LIN {X 0,Y 288.96,Z 785.854,A -85,B 0,C 180,E1 8748.983,E2 8748.983} C_VEL
LIN {X 0,Y 289.698,Z 782.109,A -85,B 0,C 180,E1 8744.907,E2 8744.907} C_VEL
LIN {X 0,Y 291.072,Z 776.715,A -85,B 0,C 180,E1 8740.892,E2 8740.892} C_VEL
LIN {X 0,Y 293.159,Z 769.854,A -85,B 0,C 180,E1 8737.044,E2 8737.044} C_VEL
LIN {X 0,Y 296.063,Z 761.342,A -85,B 0,C 180,E1 8733.293,E2 8733.293} C_VEL
LIN {X 0,Y 299.636,Z 751.536,A -85,B 0,C 180,E1 8729.811,E2 8729.811} C_VEL
LIN {X 0,Y 304.006,Z 739.719,A -85,B 0,C 180,E1 8726.419,E2 8726.419} C_VEL
LIN {X 0,Y 308.871,Z 726.48,A -85,B 0,C 180,E1 8723.31,E2 8723.31} C_VEL
LIN {X 0,Y 314.092,Z 711.806,A -85,B 0,C 180,E1 8720.474,E2 8720.474} C_VEL
LIN {X 0,Y 319.545,Z 695.592,A -85,B 0,C 180,E1 8717.901,E2 8717.901} C_VEL
LIN {X 0,Y 324.669,Z 679.065,A -85,B 0,C 180,E1 8715.739,E2 8715.739} C_VEL
LIN {X 0,Y 329.752,Z 660.963,A -85,B 0,C 180,E1 8713.804,E2 8713.804} C_VEL
LIN {X 0,Y 334.408,Z 641.774,A -85,B 0,C 180,E1 8712.156,E2 8712.156} C_VEL
LIN {X 0,Y 338.298,Z 622.744,A -85,B 0,C 180,E1 8710.851,E2 8710.851} C_VEL
LIN {X 0,Y 341.828,Z 601.532,A -85,B 0,C 180,E1 8709.727,E2 8709.727} C_VEL
LIN {X 0,Y 344.554,Z 579.645,A -85,B 0,C 180,E1 8708.89,E2 8708.89} C_VEL
LIN {X 0,Y 346.384,Z 556.456,A -85,B 0,C 180,E1 8708.295,E2 8708.295} C_VEL
LIN {X 0,Y 350.037,Z 495.768,A -85,B 0,C 180,E1 8706.999,E2 8706.999} C_VEL
LIN {X 0,Y 349.833,Z 488.203,A -85,B 0,C 180,E1 8706.711,E2 8706.711} C_VEL
LIN {X 0,Y 347.018,Z 468.467,A -85,B 0,C 180,E1 8705.501,E2 8705.501} C_VEL
LIN {X 0,Y 346.964,Z 461.961,A -85,B 0,C 180,E1 8705.269,E2 8705.269} C_VEL
LIN {X 0,Y 352.089,Z 380.587,A -85,B 0,C 180,E1 8703.525,E2 8703.525} C_VEL
LIN {X 0,Y 342.307,Z 363.806,A -85,B 0,C 180,E1 8700.718,E2 8700.718} C_VEL
LIN {X 0,Y 333.106,Z 349.419,A -85,B 0,C 180,E1 8697.824,E2 8697.824} C_VEL
LIN {X 0,Y 323.644,Z 335.645,A -85,B 0,C 180,E1 8694.496,E2 8694.496} C_VEL
LIN {X 0,Y 316.195,Z 325.679,A -85,B 0,C 180,E1 8691.572,E2 8691.572} C_VEL
LIN {X 0,Y 312.253,Z 320.486,A -85,B 0,C 180,E1 8689.859,E2 8689.859} C_VEL
LIN {X 0,Y 307.488,Z 314.479,A -85,B 0,C 180,E1 8687.657,E2 8687.657} C_VEL
LIN {X 0,Y 303.986,Z 310.183,A -85,B 0,C 180,E1 8685.875,E2 8685.875} C_VEL
LIN {X 0,Y 299.931,Z 305.159,A -85,B 0,C 180,E1 8683.632,E2 8683.632} C_VEL
LIN {X 0,Y 296.324,Z 300.805,A -85,B 0,C 180,E1 8681.4,E2 8681.4} C_VEL
LIN {X 0,Y 295.437,Z 299.331,A -85,B 0,C 180,E1 8680.523,E2 8680.523} C_VEL
LIN {X 0,Y 293.137,Z 295.553,A -85,B 0,C 180,E1 8677.627,E2 8677.627} C_VEL
LIN {X 0,Y 292.608,Z 294.29,A -85,B 0,C 180,E1 8676.723,E2 8676.723} C_VEL
LIN {X 0,Y 289.99,Z 290.354,A -85,B 0,C 180,E1 8672.728,E2 8672.728} C_VEL
LIN {X 0,Y 289.321,Z 288.803,A -85,B 0,C 180,E1 8671.221,E2 8671.221} C_VEL
LIN {X 0,Y 286.275,Z 283.926,A -85,B 0,C 180,E1 8662.778,E2 8662.778} C_VEL
LIN {X 0,Y 285.612,Z 283.017,A -85,B 0,C 180,E1 8658.786,E2 8658.786} C_VEL
LIN {X 0,Y 285.73,Z 283.102,A -85,B 0,C 180,E1 8652.94,E2 8652.94} C_VEL
LIN {X 0,Y 286.409,Z 284.215,A -85,B 0,C 180,E1 8649.037,E2 8649.037} C_VEL
LIN {X 0,Y 289.951,Z 289.598,A -85,B 0,C 180,E1 8640.38,E2 8640.38} C_VEL
LIN {X 0,Y 292.353,Z 293.977,A -85,B 0,C 180,E1 8636.273,E2 8636.273} C_VEL
LIN {X 0,Y 293.355,Z 295.125,A -85,B 0,C 180,E1 8635.11,E2 8635.11} C_VEL
LIN {X 0,Y 295.652,Z 299.397,A -85,B 0,C 180,E1 8632.028,E2 8632.028} C_VEL
LIN {X 0,Y 296.617,Z 300.723,A -85,B 0,C 180,E1 8631.078,E2 8631.078} C_VEL
LIN {X 0,Y 300.225,Z 305.323,A -85,B 0,C 180,E1 8628.764,E2 8628.764} C_VEL
LIN {X 0,Y 302.029,Z 307.444,A -85,B 0,C 180,E1 8627.718,E2 8627.718} C_VEL
LIN {X 0,Y 306.76,Z 313.199,A -85,B 0,C 180,E1 8625.222,E2 8625.222} C_VEL
LIN {X 0,Y 311.135,Z 318.616,A -85,B 0,C 180,E1 8623.139,E2 8623.139} C_VEL
LIN {X 0,Y 315.417,Z 324.086,A -85,B 0,C 180,E1 8621.23,E2 8621.23} C_VEL
LIN {X 0,Y 322.474,Z 333.247,A -85,B 0,C 180,E1 8618.394,E2 8618.394} C_VEL
LIN {X 0,Y 332.455,Z 347.118,A -85,B 0,C 180,E1 8614.813,E2 8614.813} C_VEL
LIN {X 0,Y 343.288,Z 363.412,A -85,B 0,C 180,E1 8611.371,E2 8611.371} C_VEL
LIN {X 0,Y 353.776,Z 380.644,A -85,B 0,C 180,E1 8608.38,E2 8608.38} C_VEL
LIN {X 0,Y 356.871,Z 386.273,A -85,B 0,C 180,E1 8607.544,E2 8607.544} C_VEL
LIN {X 0,Y 344.365,Z 598.77,A -85,B 0,C 180,E1 8603.126,E2 8603.126} C_VEL
LIN {X 0,Y 341.699,Z 620.996,A -85,B 0,C 180,E1 8602.442,E2 8602.442} C_VEL
LIN {X 0,Y 338.23,Z 641.686,A -85,B 0,C 180,E1 8601.567,E2 8601.567} C_VEL
LIN {X 0,Y 334.015,Z 662.2,A -85,B 0,C 180,E1 8600.424,E2 8600.424} C_VEL
LIN {X 0,Y 329.158,Z 681.971,A -85,B 0,C 180,E1 8599.009,E2 8599.009} C_VEL
LIN {X 0,Y 323.758,Z 701.072,A -85,B 0,C 180,E1 8597.305,E2 8597.305} C_VEL
LIN {X 0,Y 317.973,Z 719.569,A -85,B 0,C 180,E1 8595.285,E2 8595.285} C_VEL
LIN {X 0,Y 311.98,Z 737.297,A -85,B 0,C 180,E1 8592.921,E2 8592.921} C_VEL
LIN {X 0,Y 305.913,Z 753.989,A -85,B 0,C 180,E1 8590.201,E2 8590.201} C_VEL
LIN {X 0,Y 300.011,Z 769.739,A -85,B 0,C 180,E1 8587.098,E2 8587.098} C_VEL
LIN {X 0,Y 294.8,Z 783.662,A -85,B 0,C 180,E1 8583.793,E2 8583.793} C_VEL
LIN {X 0,Y 290.144,Z 796.44,A -85,B 0,C 180,E1 8580.12,E2 8580.12} C_VEL
LIN {X 0,Y 286.319,Z 807.649,A -85,B 0,C 180,E1 8576.17,E2 8576.17} C_VEL
LIN {X 0,Y 283.403,Z 817.534,A -85,B 0,C 180,E1 8571.892,E2 8571.892} C_VEL
LIN {X 0,Y 281.612,Z 825.183,A -85,B 0,C 180,E1 8567.776,E2 8567.776} C_VEL
LIN {X 0,Y 280.64,Z 831.149,A -85,B 0,C 180,E1 8563.598,E2 8563.598} C_VEL
LIN {X 0,Y 280.321,Z 835.68,A -85,B 0,C 180,E1 8559.234,E2 8559.234} C_VEL
LIN {X 0,Y 280.368,Z 838.327,A -85,B 0,C 180,E1 8555.318,E2 8555.318} C_VEL
LIN {X 0,Y 280.465,Z 839.49,A -85,B 0,C 180,E1 8551.428,E2 8551.428} C_VEL
LIN {X 0,Y 280.457,Z 839.377,A -85,B 0,C 180,E1 8547.955,E2 8547.955} C_VEL
LIN {X 0,Y 280.349,Z 837.945,A -85,B 0,C 180,E1 8544.061,E2 8544.061} C_VEL
LIN {X 0,Y 280.337,Z 835.069,A -85,B 0,C 180,E1 8540.14,E2 8540.14} C_VEL
LIN {X 0,Y 280.737,Z 830.298,A -85,B 0,C 180,E1 8535.772,E2 8535.772} C_VEL
LIN {X 0,Y 281.821,Z 824.143,A -85,B 0,C 180,E1 8531.591,E2 8531.591} C_VEL
LIN {X 0,Y 283.811,Z 816.119,A -85,B 0,C 180,E1 8527.374,E2 8527.374} C_VEL
LIN {X 0,Y 286.968,Z 805.984,A -85,B 0,C 180,E1 8523.065,E2 8523.065} C_VEL
LIN {X 0,Y 290.951,Z 794.89,A -85,B 0,C 180,E1 8519.198,E2 8519.198} C_VEL
LIN {X 0,Y 296.028,Z 781.655,A -85,B 0,C 180,E1 8515.427,E2 8515.427} C_VEL
LIN {X 0,Y 301.627,Z 767.471,A -85,B 0,C 180,E1 8512.088,E2 8512.088} C_VEL
LIN {X 0,Y 308.077,Z 751.16,A -85,B 0,C 180,E1 8508.91,E2 8508.91} C_VEL
LIN {X 0,Y 314.475,Z 734.51,A -85,B 0,C 180,E1 8506.234,E2 8506.234} C_VEL
LIN {X 0,Y 320.933,Z 716.552,A -85,B 0,C 180,E1 8503.876,E2 8503.876} C_VEL
LIN {X 0,Y 327.063,Z 698.101,A -85,B 0,C 180,E1 8501.891,E2 8501.891} C_VEL
LIN {X 0,Y 332.717,Z 679.347,A -85,B 0,C 180,E1 8500.242,E2 8500.242} C_VEL
LIN {X 0,Y 338.053,Z 658.99,A -85,B 0,C 180,E1 8498.81,E2 8498.81} C_VEL
LIN {X 0,Y 342.508,Z 638.773,A -85,B 0,C 180,E1 8497.709,E2 8497.709} C_VEL
LIN {X 0,Y 346.488,Z 616.391,A -85,B 0,C 180,E1 8496.8,E2 8496.8} C_VEL
LIN {X 0,Y 349.201,Z 594.573,A -85,B 0,C 180,E1 8496.155,E2 8496.155} C_VEL
LIN {X 0,Y 363.212,Z 387.306,A -85,B 0,C 180,E1 8491.769,E2 8491.769} C_VEL
LIN {X 0,Y 357.13,Z 375.817,A -85,B 0,C 180,E1 8489.469,E2 8489.469} C_VEL
LIN {X 0,Y 351.809,Z 366.536,A -85,B 0,C 180,E1 8487.179,E2 8487.179} C_VEL
LIN {X 0,Y 346.722,Z 358.345,A -85,B 0,C 180,E1 8484.628,E2 8484.628} C_VEL
LIN {X 0,Y 342.725,Z 352.195,A -85,B 0,C 180,E1 8482.199,E2 8482.199} C_VEL
LIN {X 0,Y 338.782,Z 346.281,A -85,B 0,C 180,E1 8479.124,E2 8479.124} C_VEL
LIN {X 0,Y 335.351,Z 341.275,A -85,B 0,C 180,E1 8474.858,E2 8474.858} C_VEL
LIN {X 0,Y 334.083,Z 340.173,A -85,B 0,C 180,E1 8470.869,E2 8470.869} C_VEL
LIN {X 0,Y 334.8,Z 340.86,A -85,B 0,C 180,E1 8467.034,E2 8467.034} C_VEL
LIN {X 0,Y 335.429,Z 341.751,A -85,B 0,C 180,E1 8465.732,E2 8465.732} C_VEL
LIN {X 0,Y 338.722,Z 346.674,A -85,B 0,C 180,E1 8461.693,E2 8461.693} C_VEL
LIN {X 0,Y 342.538,Z 352.567,A -85,B 0,C 180,E1 8458.663,E2 8458.663} C_VEL
LIN {X 0,Y 346.974,Z 359.516,A -85,B 0,C 180,E1 8455.953,E2 8455.953} C_VEL
LIN {X 0,Y 351.61,Z 367.232,A -85,B 0,C 180,E1 8453.593,E2 8453.593} C_VEL
LIN {X 0,Y 357.61,Z 377.851,A -85,B 0,C 180,E1 8450.993,E2 8450.993} C_VEL
LIN {X 0,Y 361.836,Z 386.289,A -85,B 0,C 180,E1 8449.342,E2 8449.342} C_VEL
LIN {X 0,Y 347.156,Z 576.519,A -85,B 0,C 180,E1 8445.157,E2 8445.157} C_VEL
LIN {X 0,Y 344.505,Z 597.249,A -85,B 0,C 180,E1 8444.439,E2 8444.439} C_VEL
LIN {X 0,Y 341.005,Z 617.374,A -85,B 0,C 180,E1 8443.478,E2 8443.478} C_VEL
LIN {X 0,Y 336.446,Z 638.132,A -85,B 0,C 180,E1 8442.178,E2 8442.178} C_VEL
LIN {X 0,Y 331.586,Z 656.641,A -85,B 0,C 180,E1 8440.706,E2 8440.706} C_VEL
LIN {X 0,Y 325.902,Z 675.297,A -85,B 0,C 180,E1 8438.857,E2 8438.857} C_VEL
LIN {X 0,Y 319.749,Z 693.072,A -85,B 0,C 180,E1 8436.667,E2 8436.667} C_VEL
LIN {X 0,Y 313.63,Z 709.09,A -85,B 0,C 180,E1 8434.242,E2 8434.242} C_VEL
LIN {X 0,Y 307.613,Z 723.755,A -85,B 0,C 180,E1 8431.533,E2 8431.533} C_VEL
LIN {X 0,Y 301.449,Z 738.039,A -85,B 0,C 180,E1 8428.298,E2 8428.298} C_VEL
LIN {X 0,Y 296.18,Z 749.926,A -85,B 0,C 180,E1 8424.98,E2 8424.98} C_VEL
LIN {X 0,Y 291.545,Z 760.386,A -85,B 0,C 180,E1 8421.381,E2 8421.381} C_VEL
LIN {X 0,Y 287.493,Z 769.777,A -85,B 0,C 180,E1 8417.301,E2 8417.301} C_VEL
LIN {X 0,Y 284.581,Z 776.948,A -85,B 0,C 180,E1 8413.247,E2 8413.247} C_VEL
LIN {X 0,Y 282.636,Z 782.301,A -85,B 0,C 180,E1 8409.223,E2 8409.223} C_VEL
LIN {X 0,Y 281.403,Z 786.349,A -85,B 0,C 180,E1 8404.842,E2 8404.842} C_VEL
LIN {X 0,Y 280.867,Z 788.559,A -85,B 0,C 180,E1 8400.841,E2 8400.841} C_VEL
LIN {X 0,Y 280.669,Z 789.27,A -85,B 0,C 180,E1 8396.902,E2 8396.902} C_VEL
LIN {X 0,Y 280.703,Z 788.609,A -85,B 0,C 180,E1 8392.848,E2 8392.848} C_VEL
LIN {X 0,Y 281.012,Z 786.58,A -85,B 0,C 180,E1 8388.844,E2 8388.844} C_VEL
LIN {X 0,Y 281.762,Z 782.987,A -85,B 0,C 180,E1 8384.805,E2 8384.805} C_VEL
LIN {X 0,Y 283.151,Z 777.829,A -85,B 0,C 180,E1 8380.789,E2 8380.789} C_VEL
LIN {X 0,Y 285.445,Z 770.71,A -85,B 0,C 180,E1 8376.64,E2 8376.64} C_VEL
LIN {X 0,Y 288.513,Z 762.206,A -85,B 0,C 180,E1 8372.783,E2 8372.783} C_VEL
LIN {X 0,Y 292.494,Z 751.817,A -85,B 0,C 180,E1 8369.023,E2 8369.023} C_VEL
LIN {X 0,Y 297.12,Z 739.943,A -85,B 0,C 180,E1 8365.563,E2 8365.563} C_VEL
LIN {X 0,Y 302.24,Z 726.611,A -85,B 0,C 180,E1 8362.398,E2 8362.398} C_VEL
LIN {X 0,Y 307.541,Z 712.321,A -85,B 0,C 180,E1 8359.607,E2 8359.607} C_VEL
LIN {X 0,Y 313.218,Z 696.066,A -85,B 0,C 180,E1 8356.996,E2 8356.996} C_VEL
LIN {X 0,Y 318.548,Z 679.49,A -85,B 0,C 180,E1 8354.808,E2 8354.808} C_VEL
LIN {X 0,Y 323.823,Z 661.34,A -85,B 0,C 180,E1 8352.852,E2 8352.852} C_VEL
LIN {X 0,Y 328.65,Z 642.115,A -85,B 0,C 180,E1 8351.189,E2 8351.189} C_VEL
LIN {X 0,Y 332.677,Z 623.038,A -85,B 0,C 180,E1 8349.874,E2 8349.874} C_VEL
LIN {X 0,Y 336.314,Z 601.867,A -85,B 0,C 180,E1 8348.747,E2 8348.747} C_VEL
LIN {X 0,Y 339.148,Z 579.793,A -85,B 0,C 180,E1 8347.9,E2 8347.9} C_VEL
LIN {X 0,Y 341.054,Z 556.224,A -85,B 0,C 180,E1 8347.295,E2 8347.295} C_VEL
LIN {X 0,Y 346.964,Z 461.961,A -85,B 0,C 180,E1 8345.269,E2 8345.269} C_VEL
LIN {X 0,Y 346.834,Z 454.394,A -85,B 0,C 180,E1 8344.982,E2 8344.982} C_VEL
LIN {X 0,Y 344.217,Z 434.656,A -85,B 0,C 180,E1 8343.751,E2 8343.751} C_VEL
LIN {X 0,Y 344.179,Z 428.151,A -85,B 0,C 180,E1 8343.512,E2 8343.512} C_VEL
LIN {X 0,Y 346.995,Z 384.26,A -85,B 0,C 180,E1 8342.555,E2 8342.555} C_VEL
LIN {X 0,Y 337.233,Z 367.447,A -85,B 0,C 180,E1 8339.626,E2 8339.626} C_VEL
LIN {X 0,Y 328.644,Z 354.039,A -85,B 0,C 180,E1 8336.798,E2 8336.798} C_VEL
LIN {X 0,Y 320.15,Z 341.516,A -85,B 0,C 180,E1 8333.68,E2 8333.68} C_VEL
LIN {X 0,Y 313.353,Z 332.296,A -85,B 0,C 180,E1 8330.908,E2 8330.908} C_VEL
LIN {X 0,Y 309.764,Z 327.505,A -85,B 0,C 180,E1 8329.309,E2 8329.309} C_VEL
LIN {X 0,Y 304.951,Z 321.32,A -85,B 0,C 180,E1 8327.005,E2 8327.005} C_VEL
LIN {X 0,Y 301.631,Z 317.18,A -85,B 0,C 180,E1 8325.248,E2 8325.248} C_VEL
LIN {X 0,Y 297.992,Z 312.599,A -85,B 0,C 180,E1 8323.192,E2 8323.192} C_VEL
LIN {X 0,Y 294.364,Z 308.114,A -85,B 0,C 180,E1 8320.895,E2 8320.895} C_VEL
LIN {X 0,Y 292.939,Z 306.545,A -85,B 0,C 180,E1 8319.914,E2 8319.914} C_VEL
LIN {X 0,Y 289.269,Z 302.244,A -85,B 0,C 180,E1 8317.218,E2 8317.218} C_VEL
LIN {X 0,Y 288.179,Z 300.837,A -85,B 0,C 180,E1 8316.265,E2 8316.265} C_VEL
LIN {X 0,Y 285.556,Z 296.562,A -85,B 0,C 180,E1 8312.153,E2 8312.153} C_VEL
LIN {X 0,Y 284.77,Z 295.304,A -85,B 0,C 180,E1 8310.602,E2 8310.602} C_VEL
LIN {X 0,Y 282.142,Z 290.71,A -85,B 0,C 180,E1 8302.501,E2 8302.501} C_VEL
LIN {X 0,Y 281.507,Z 289.878,A -85,B 0,C 180,E1 8298.211,E2 8298.211} C_VEL
LIN {X 0,Y 281.76,Z 290.08,A -85,B 0,C 180,E1 8292.5,E2 8292.5} C_VEL
LIN {X 0,Y 282.36,Z 291.206,A -85,B 0,C 180,E1 8288.917,E2 8288.917} C_VEL
LIN {X 0,Y 285.744,Z 296.313,A -85,B 0,C 180,E1 8280.6,E2 8280.6} C_VEL
LIN {X 0,Y 288.201,Z 300.781,A -85,B 0,C 180,E1 8276.418,E2 8276.418} C_VEL
LIN {X 0,Y 289.496,Z 302.21,A -85,B 0,C 180,E1 8275.244,E2 8275.244} C_VEL
LIN {X 0,Y 293.06,Z 306.64,A -85,B 0,C 180,E1 8272.549,E2 8272.549} C_VEL
LIN {X 0,Y 294.752,Z 308.37,A -85,B 0,C 180,E1 8271.415,E2 8271.415} C_VEL
LIN {X 0,Y 298.672,Z 313.092,A -85,B 0,C 180,E1 8268.998,E2 8268.998} C_VEL
LIN {X 0,Y 304.696,Z 320.601,A -85,B 0,C 180,E1 8265.654,E2 8265.654} C_VEL
LIN {X 0,Y 308.931,Z 325.927,A -85,B 0,C 180,E1 8263.596,E2 8263.596} C_VEL
LIN {X 0,Y 313.153,Z 331.425,A -85,B 0,C 180,E1 8261.668,E2 8261.668} C_VEL
LIN {X 0,Y 319.919,Z 340.337,A -85,B 0,C 180,E1 8258.887,E2 8258.887} C_VEL
LIN {X 0,Y 329.429,Z 353.77,A -85,B 0,C 180,E1 8255.381,E2 8255.381} C_VEL
LIN {X 0,Y 339.989,Z 369.918,A -85,B 0,C 180,E1 8251.93,E2 8251.93} C_VEL
LIN {X 0,Y 350.662,Z 387.725,A -85,B 0,C 180,E1 8248.809,E2 8248.809} C_VEL
LIN {X 0,Y 351.752,Z 389.961,A -85,B 0,C 180,E1 8248.496,E2 8248.496} C_VEL
LIN {X 0,Y 339.052,Z 598.328,A -85,B 0,C 180,E1 8244.137,E2 8244.137} C_VEL
LIN {X 0,Y 336.324,Z 620.453,A -85,B 0,C 180,E1 8243.455,E2 8243.455} C_VEL
LIN {X 0,Y 332.728,Z 641.297,A -85,B 0,C 180,E1 8242.572,E2 8242.572} C_VEL
LIN {X 0,Y 328.51,Z 661.261,A -85,B 0,C 180,E1 8241.459,E2 8241.459} C_VEL
LIN {X 0,Y 323.497,Z 681.072,A -85,B 0,C 180,E1 8240.038,E2 8240.038} C_VEL
LIN {X 0,Y 317.936,Z 700.164,A -85,B 0,C 180,E1 8238.332,E2 8238.332} C_VEL
LIN {X 0,Y 311.912,Z 718.8,A -85,B 0,C 180,E1 8236.287,E2 8236.287} C_VEL
LIN {X 0,Y 305.677,Z 736.578,A -85,B 0,C 180,E1 8233.9,E2 8233.9} C_VEL
LIN {X 0,Y 299.5,Z 752.941,A -85,B 0,C 180,E1 8231.209,E2 8231.209} C_VEL
LIN {X 0,Y 293.274,Z 768.84,A -85,B 0,C 180,E1 8228.042,E2 8228.042} C_VEL
LIN {X 0,Y 287.866,Z 782.632,A -85,B 0,C 180,E1 8224.721,E2 8224.721} C_VEL
LIN {X 0,Y 283.011,Z 795.216,A -85,B 0,C 180,E1 8221.049,E2 8221.049} C_VEL
LIN {X 0,Y 278.97,Z 806.37,A -85,B 0,C 180,E1 8217.074,E2 8217.074} C_VEL
LIN {X 0,Y 275.752,Z 816.549,A -85,B 0,C 180,E1 8212.601,E2 8212.601} C_VEL
LIN {X 0,Y 273.762,Z 824.423,A -85,B 0,C 180,E1 8208.266,E2 8208.266} C_VEL
LIN {X 0,Y 272.705,Z 830.359,A -85,B 0,C 180,E1 8204.001,E2 8204.001} C_VEL
LIN {X 0,Y 272.344,Z 834.925,A -85,B 0,C 180,E1 8199.507,E2 8199.507} C_VEL
LIN {X 0,Y 272.381,Z 837.47,A -85,B 0,C 180,E1 8195.686,E2 8195.686} C_VEL
LIN {X 0,Y 272.492,Z 838.748,A -85,B 0,C 180,E1 8191.68,E2 8191.68} C_VEL
LIN {X 0,Y 272.491,Z 838.693,A -85,B 0,C 180,E1 8188.105,E2 8188.105} C_VEL
LIN {X 0,Y 272.372,Z 837.365,A -85,B 0,C 180,E1 8184.098,E2 8184.098} C_VEL
LIN {X 0,Y 272.352,Z 834.541,A -85,B 0,C 180,E1 8180.062,E2 8180.062} C_VEL
LIN {X 0,Y 272.771,Z 829.868,A -85,B 0,C 180,E1 8175.564,E2 8175.564} C_VEL
LIN {X 0,Y 273.914,Z 823.762,A -85,B 0,C 180,E1 8171.261,E2 8171.261} C_VEL
LIN {X 0,Y 276.007,Z 815.908,A -85,B 0,C 180,E1 8166.948,E2 8166.948} C_VEL
LIN {X 0,Y 279.251,Z 806.144,A -85,B 0,C 180,E1 8162.62,E2 8162.62} C_VEL
LIN {X 0,Y 283.549,Z 794.847,A -85,B 0,C 180,E1 8158.539,E2 8158.539} C_VEL
LIN {X 0,Y 288.869,Z 781.727,A -85,B 0,C 180,E1 8154.685,E2 8154.685} C_VEL
LIN {X 0,Y 294.968,Z 767.163,A -85,B 0,C 180,E1 8151.162,E2 8151.162} C_VEL
LIN {X 0,Y 301.446,Z 751.617,A -85,B 0,C 180,E1 8148.058,E2 8148.058} C_VEL
LIN {X 0,Y 308.373,Z 734.455,A -85,B 0,C 180,E1 8145.243,E2 8145.243} C_VEL
LIN {X 0,Y 315.108,Z 716.565,A -85,B 0,C 180,E1 8142.861,E2 8142.861} C_VEL
LIN {X 0,Y 321.655,Z 697.65,A -85,B 0,C 180,E1 8140.805,E2 8140.805} C_VEL
LIN {X 0,Y 327.521,Z 679.016,A -85,B 0,C 180,E1 8139.155,E2 8139.155} C_VEL
LIN {X 0,Y 333.072,Z 658.633,A -85,B 0,C 180,E1 8137.718,E2 8137.718} C_VEL
LIN {X 0,Y 337.797,Z 637.894,A -85,B 0,C 180,E1 8136.592,E2 8136.592} C_VEL
LIN {X 0,Y 341.94,Z 615.26,A -85,B 0,C 180,E1 8135.683,E2 8135.683} C_VEL
LIN {X 0,Y 344.716,Z 593.311,A -85,B 0,C 180,E1 8135.039,E2 8135.039} C_VEL
LIN {X 0,Y 358.984,Z 391.402,A -85,B 0,C 180,E1 8130.738,E2 8130.738} C_VEL
LIN {X 0,Y 353.499,Z 380.693,A -85,B 0,C 180,E1 8128.51,E2 8128.51} C_VEL
LIN {X 0,Y 347.702,Z 370.44,A -85,B 0,C 180,E1 8125.782,E2 8125.782} C_VEL
LIN {X 0,Y 342.941,Z 362.606,A -85,B 0,C 180,E1 8123.089,E2 8123.089} C_VEL
LIN {X 0,Y 339.712,Z 357.776,A -85,B 0,C 180,E1 8120.864,E2 8120.864} C_VEL
LIN {X 0,Y 337.208,Z 353.82,A -85,B 0,C 180,E1 8118.678,E2 8118.678} C_VEL
LIN {X 0,Y 334.208,Z 349.161,A -85,B 0,C 180,E1 8114.733,E2 8114.733} C_VEL
LIN {X 0,Y 333.004,Z 348.094,A -85,B 0,C 180,E1 8110.73,E2 8110.73} C_VEL
LIN {X 0,Y 333.784,Z 348.857,A -85,B 0,C 180,E1 8106.883,E2 8106.883} C_VEL
LIN {X 0,Y 334.321,Z 349.825,A -85,B 0,C 180,E1 8105.751,E2 8105.751} C_VEL
LIN {X 0,Y 337.323,Z 354.442,A -85,B 0,C 180,E1 8101.955,E2 8101.955} C_VEL
LIN {X 0,Y 341.021,Z 360.377,A -85,B 0,C 180,E1 8098.899,E2 8098.899} C_VEL
LIN {X 0,Y 345.256,Z 367.344,A -85,B 0,C 180,E1 8096.224,E2 8096.224} C_VEL
LIN {X 0,Y 349.539,Z 374.718,A -85,B 0,C 180,E1 8093.967,E2 8093.967} C_VEL
LIN {X 0,Y 355.163,Z 385.134,A -85,B 0,C 180,E1 8091.421,E2 8091.421} C_VEL
LIN {X 0,Y 357.679,Z 390.488,A -85,B 0,C 180,E1 8090.376,E2 8090.376} C_VEL
LIN {X 0,Y 342.678,Z 577.001,A -85,B 0,C 180,E1 8086.256,E2 8086.256} C_VEL
LIN {X 0,Y 339.89,Z 597.985,A -85,B 0,C 180,E1 8085.526,E2 8085.526} C_VEL
LIN {X 0,Y 336.338,Z 617.732,A -85,B 0,C 180,E1 8084.583,E2 8084.583} C_VEL
LIN {X 0,Y 331.695,Z 638.196,A -85,B 0,C 180,E1 8083.304,E2 8083.304} C_VEL
LIN {X 0,Y 326.543,Z 657.073,A -85,B 0,C 180,E1 8081.803,E2 8081.803} C_VEL
LIN {X 0,Y 320.484,Z 676.157,A -85,B 0,C 180,E1 8079.9,E2 8079.9} C_VEL
LIN {X 0,Y 314.241,Z 693.465,A -85,B 0,C 180,E1 8077.753,E2 8077.753} C_VEL
LIN {X 0,Y 307.989,Z 709.12,A -85,B 0,C 180,E1 8075.37,E2 8075.37} C_VEL
LIN {X 0,Y 301.488,Z 724.292,A -85,B 0,C 180,E1 8072.552,E2 8072.552} C_VEL
LIN {X 0,Y 295.167,Z 738.222,A -85,B 0,C 180,E1 8069.365,E2 8069.365} C_VEL
LIN {X 0,Y 289.548,Z 750.249,A -85,B 0,C 180,E1 8065.974,E2 8065.974} C_VEL
LIN {X 0,Y 284.531,Z 760.916,A -85,B 0,C 180,E1 8062.25,E2 8062.25} C_VEL
LIN {X 0,Y 280.248,Z 770.153,A -85,B 0,C 180,E1 8058.154,E2 8058.154} C_VEL
LIN {X 0,Y 277.155,Z 777.214,A -85,B 0,C 180,E1 8054.121,E2 8054.121} C_VEL
LIN {X 0,Y 274.913,Z 782.902,A -85,B 0,C 180,E1 8049.802,E2 8049.802} C_VEL
LIN {X 0,Y 273.568,Z 786.914,A -85,B 0,C 180,E1 8045.413,E2 8045.413} C_VEL
LIN {X 0,Y 272.932,Z 789.272,A -85,B 0,C 180,E1 8041.103,E2 8041.103} C_VEL
LIN {X 0,Y 272.704,Z 789.991,A -85,B 0,C 180,E1 8037.013,E2 8037.013} C_VEL
LIN {X 0,Y 272.735,Z 789.349,A -85,B 0,C 180,E1 8032.87,E2 8032.87} C_VEL
LIN {X 0,Y 273.055,Z 787.381,A -85,B 0,C 180,E1 8028.8,E2 8028.8} C_VEL
LIN {X 0,Y 273.855,Z 783.757,A -85,B 0,C 180,E1 8024.593,E2 8024.593} C_VEL
LIN {X 0,Y 275.398,Z 778.411,A -85,B 0,C 180,E1 8020.313,E2 8020.313} C_VEL
LIN {X 0,Y 277.901,Z 771.131,A -85,B 0,C 180,E1 8015.991,E2 8015.991} C_VEL
LIN {X 0,Y 281.18,Z 762.557,A -85,B 0,C 180,E1 8012.04,E2 8012.04} C_VEL
LIN {X 0,Y 285.166,Z 752.713,A -85,B 0,C 180,E1 8008.395,E2 8008.395} C_VEL
LIN {X 0,Y 290.159,Z 740.486,A -85,B 0,C 180,E1 8004.759,E2 8004.759} C_VEL
LIN {X 0,Y 295.347,Z 727.548,A -85,B 0,C 180,E1 8001.632,E2 8001.632} C_VEL
LIN {X 0,Y 301.057,Z 712.802,A -85,B 0,C 180,E1 7998.702,E2 7998.702} C_VEL
LIN {X 0,Y 307.022,Z 696.365,A -85,B 0,C 180,E1 7996.033,E2 7996.033} C_VEL
LIN {X 0,Y 312.734,Z 679.185,A -85,B 0,C 180,E1 7993.757,E2 7993.757} C_VEL
LIN {X 0,Y 317.989,Z 661.713,A -85,B 0,C 180,E1 7991.865,E2 7991.865} C_VEL
LIN {X 0,Y 323.014,Z 642.356,A -85,B 0,C 180,E1 7990.18,E2 7990.18} C_VEL
LIN {X 0,Y 327.155,Z 623.318,A -85,B 0,C 180,E1 7988.863,E2 7988.863} C_VEL
LIN {X 0,Y 330.883,Z 602.263,A -85,B 0,C 180,E1 7987.739,E2 7987.739} C_VEL
LIN {X 0,Y 333.807,Z 580.158,A -85,B 0,C 180,E1 7986.887,E2 7986.887} C_VEL
LIN {X 0,Y 335.784,Z 556.475,A -85,B 0,C 180,E1 7986.276,E2 7986.276} C_VEL
LIN {X 0,Y 344.179,Z 428.151,A -85,B 0,C 180,E1 7983.512,E2 7983.512} C_VEL
LIN {X 0,Y 344.071,Z 420.587,A -85,B 0,C 180,E1 7983.219,E2 7983.219} C_VEL
LIN {X 0,Y 341.681,Z 400.852,A -85,B 0,C 180,E1 7981.965,E2 7981.965} C_VEL
LIN {X 0,Y 341.691,Z 394.348,A -85,B 0,C 180,E1 7981.725,E2 7981.725} C_VEL
LIN {X 0,Y 342.005,Z 387.904,A -85,B 0,C 180,E1 7981.556,E2 7981.556} C_VEL
LIN {X 0,Y 332.733,Z 371.977,A -85,B 0,C 180,E1 7978.656,E2 7978.656} C_VEL
LIN {X 0,Y 324.252,Z 358.492,A -85,B 0,C 180,E1 7975.727,E2 7975.727} C_VEL
LIN {X 0,Y 315.231,Z 345.305,A -85,B 0,C 180,E1 7972.243,E2 7972.243} C_VEL
LIN {X 0,Y 307.973,Z 335.301,A -85,B 0,C 180,E1 7969.061,E2 7969.061} C_VEL
LIN {X 0,Y 302.234,Z 327.866,A -85,B 0,C 180,E1 7966.225,E2 7966.225} C_VEL
LIN {X 0,Y 296.244,Z 320.199,A -85,B 0,C 180,E1 7962.847,E2 7962.847} C_VEL
LIN {X 0,Y 292.529,Z 315.531,A -85,B 0,C 180,E1 7960.424,E2 7960.424} C_VEL
LIN {X 0,Y 287.612,Z 309.77,A -85,B 0,C 180,E1 7956.782,E2 7956.782} C_VEL
LIN {X 0,Y 286.446,Z 308.361,A -85,B 0,C 180,E1 7955.777,E2 7955.777} C_VEL
LIN {X 0,Y 282.685,Z 304.219,A -85,B 0,C 180,E1 7952.16,E2 7952.16} C_VEL
LIN {X 0,Y 281.462,Z 302.631,A -85,B 0,C 180,E1 7950.725,E2 7950.725} C_VEL
LIN {X 0,Y 278.356,Z 298.664,A -85,B 0,C 180,E1 7944.622,E2 7944.622} C_VEL
LIN {X 0,Y 277.809,Z 297.122,A -85,B 0,C 180,E1 7941.092,E2 7941.092} C_VEL
LIN {X 0,Y 277.397,Z 296.702,A -85,B 0,C 180,E1 7935.253,E2 7935.253} C_VEL
LIN {X 0,Y 278.092,Z 297.479,A -85,B 0,C 180,E1 7930.355,E2 7930.355} C_VEL
LIN {X 0,Y 280.41,Z 301.707,A -85,B 0,C 180,E1 7923.269,E2 7923.269} C_VEL
LIN {X 0,Y 282.636,Z 303.83,A -85,B 0,C 180,E1 7920.606,E2 7920.606} C_VEL
LIN {X 0,Y 286.242,Z 308.201,A -85,B 0,C 180,E1 7916.995,E2 7916.995} C_VEL
LIN {X 0,Y 287.905,Z 309.861,A -85,B 0,C 180,E1 7915.617,E2 7915.617} C_VEL
LIN {X 0,Y 291.578,Z 314.393,A -85,B 0,C 180,E1 7912.808,E2 7912.808} C_VEL
LIN {X 0,Y 293.091,Z 316.06,A -85,B 0,C 180,E1 7911.761,E2 7911.761} C_VEL
LIN {X 0,Y 297.114,Z 320.857,A -85,B 0,C 180,E1 7909.234,E2 7909.234} C_VEL
LIN {X 0,Y 302.904,Z 328.34,A -85,B 0,C 180,E1 7905.958,E2 7905.958} C_VEL
LIN {X 0,Y 306.747,Z 333.244,A -85,B 0,C 180,E1 7904.054,E2 7904.054} C_VEL
LIN {X 0,Y 311.002,Z 338.889,A -85,B 0,C 180,E1 7902.07,E2 7902.07} C_VEL
LIN {X 0,Y 317.354,Z 347.416,A -85,B 0,C 180,E1 7899.384,E2 7899.384} C_VEL
LIN {X 0,Y 326.523,Z 360.593,A -85,B 0,C 180,E1 7895.918,E2 7895.918} C_VEL
LIN {X 0,Y 336.608,Z 376.224,A -85,B 0,C 180,E1 7892.537,E2 7892.537} C_VEL
LIN {X 0,Y 346.734,Z 393.391,A -85,B 0,C 180,E1 7889.482,E2 7889.482} C_VEL
LIN {X 0,Y 333.782,Z 598.044,A -85,B 0,C 180,E1 7885.168,E2 7885.168} C_VEL
LIN {X 0,Y 330.97,Z 620.222,A -85,B 0,C 180,E1 7884.481,E2 7884.481} C_VEL
LIN {X 0,Y 327.145,Z 641.675,A -85,B 0,C 180,E1 7883.565,E2 7883.565} C_VEL
LIN {X 0,Y 322.611,Z 662.247,A -85,B 0,C 180,E1 7882.397,E2 7882.397} C_VEL
LIN {X 0,Y 317.397,Z 682.169,A -85,B 0,C 180,E1 7880.946,E2 7880.946} C_VEL
LIN {X 0,Y 311.634,Z 701.086,A -85,B 0,C 180,E1 7879.214,E2 7879.214} C_VEL
LIN {X 0,Y 305.052,Z 720.489,A -85,B 0,C 180,E1 7877.018,E2 7877.018} C_VEL
LIN {X 0,Y 298.777,Z 737.598,A -85,B 0,C 180,E1 7874.646,E2 7874.646} C_VEL
LIN {X 0,Y 292.265,Z 754.161,A -85,B 0,C 180,E1 7871.841,E2 7871.841} C_VEL
LIN {X 0,Y 286.065,Z 769.269,A -85,B 0,C 180,E1 7868.726,E2 7868.726} C_VEL
LIN {X 0,Y 280.074,Z 783.801,A -85,B 0,C 180,E1 7865.08,E2 7865.08} C_VEL
LIN {X 0,Y 275.107,Z 796.156,A -85,B 0,C 180,E1 7861.311,E2 7861.311} C_VEL
LIN {X 0,Y 270.973,Z 807.083,A -85,B 0,C 180,E1 7857.217,E2 7857.217} C_VEL
LIN {X 0,Y 267.834,Z 816.54,A -85,B 0,C 180,E1 7852.843,E2 7852.843} C_VEL
LIN {X 0,Y 265.719,Z 824.52,A -85,B 0,C 180,E1 7848.196,E2 7848.196} C_VEL
LIN {X 0,Y 264.671,Z 830.371,A -85,B 0,C 180,E1 7843.766,E2 7843.766} C_VEL
LIN {X 0,Y 264.358,Z 834.505,A -85,B 0,C 180,E1 7839.357,E2 7839.357} C_VEL
LIN {X 0,Y 264.425,Z 837.071,A -85,B 0,C 180,E1 7835.204,E2 7835.204} C_VEL
LIN {X 0,Y 264.532,Z 838.069,A -85,B 0,C 180,E1 7831.297,E2 7831.297} C_VEL
LIN {X 0,Y 264.509,Z 837.913,A -85,B 0,C 180,E1 7827.615,E2 7827.615} C_VEL
LIN {X 0,Y 264.384,Z 836.402,A -85,B 0,C 180,E1 7823.483,E2 7823.483} C_VEL
LIN {X 0,Y 264.393,Z 833.467,A -85,B 0,C 180,E1 7819.319,E2 7819.319} C_VEL
LIN {X 0,Y 264.93,Z 828.606,A -85,B 0,C 180,E1 7814.679,E2 7814.679} C_VEL
LIN {X 0,Y 266.28,Z 822.397,A -85,B 0,C 180,E1 7810.246,E2 7810.246} C_VEL
LIN {X 0,Y 268.8,Z 813.94,A -85,B 0,C 180,E1 7805.611,E2 7805.611} C_VEL
LIN {X 0,Y 272.404,Z 804.078,A -85,B 0,C 180,E1 7801.258,E2 7801.258} C_VEL
LIN {X 0,Y 276.996,Z 792.902,A -85,B 0,C 180,E1 7797.216,E2 7797.216} C_VEL
LIN {X 0,Y 282.752,Z 779.637,A -85,B 0,C 180,E1 7793.299,E2 7793.299} C_VEL
LIN {X 0,Y 289.051,Z 765.372,A -85,B 0,C 180,E1 7789.861,E2 7789.861} C_VEL
LIN {X 0,Y 296.203,Z 748.987,A -85,B 0,C 180,E1 7786.61,E2 7786.61} C_VEL
LIN {X 0,Y 303.218,Z 732.295,A -85,B 0,C 180,E1 7783.902,E2 7783.902} C_VEL
LIN {X 0,Y 310.38,Z 714.079,A -85,B 0,C 180,E1 7781.496,E2 7781.496} C_VEL
LIN {X 0,Y 316.94,Z 695.667,A -85,B 0,C 180,E1 7779.524,E2 7779.524} C_VEL
LIN {X 0,Y 323.332,Z 675.695,A -85,B 0,C 180,E1 7777.803,E2 7777.803} C_VEL
LIN {X 0,Y 328.815,Z 656.148,A -85,B 0,C 180,E1 7776.456,E2 7776.456} C_VEL
LIN {X 0,Y 333.73,Z 634.966,A -85,B 0,C 180,E1 7775.342,E2 7775.342} C_VEL
LIN {X 0,Y 337.671,Z 613.515,A -85,B 0,C 180,E1 7774.51,E2 7774.51} C_VEL
LIN {X 0,Y 340.511,Z 590.706,A -85,B 0,C 180,E1 7773.859,E2 7773.859} C_VEL
LIN {X 0,Y 354.96,Z 395.509,A -85,B 0,C 180,E1 7769.69,E2 7769.69} C_VEL
LIN {X 0,Y 349.664,Z 385.109,A -85,B 0,C 180,E1 7767.366,E2 7767.366} C_VEL
LIN {X 0,Y 344.967,Z 376.662,A -85,B 0,C 180,E1 7764.99,E2 7764.99} C_VEL
LIN {X 0,Y 340.877,Z 369.622,A -85,B 0,C 180,E1 7762.507,E2 7762.507} C_VEL
LIN {X 0,Y 338.036,Z 365.197,A -85,B 0,C 180,E1 7760.429,E2 7760.429} C_VEL
LIN {X 0,Y 335.83,Z 361.54,A -85,B 0,C 180,E1 7758.398,E2 7758.398} C_VEL
LIN {X 0,Y 332.977,Z 356.966,A -85,B 0,C 180,E1 7754.433,E2 7754.433} C_VEL
LIN {X 0,Y 331.928,Z 356.012,A -85,B 0,C 180,E1 7750.414,E2 7750.414} C_VEL
LIN {X 0,Y 332.904,Z 356.986,A -85,B 0,C 180,E1 7746.468,E2 7746.468} C_VEL
LIN {X 0,Y 335.93,Z 362.207,A -85,B 0,C 180,E1 7742.219,E2 7742.219} C_VEL
LIN {X 0,Y 339.259,Z 367.758,A -85,B 0,C 180,E1 7739.326,E2 7739.326} C_VEL
LIN {X 0,Y 343.266,Z 374.648,A -85,B 0,C 180,E1 7736.662,E2 7736.662} C_VEL
LIN {X 0,Y 347.492,Z 382.202,A -85,B 0,C 180,E1 7734.342,E2 7734.342} C_VEL
LIN {X 0,Y 352.851,Z 392.593,A -85,B 0,C 180,E1 7731.815,E2 7731.815} C_VEL
LIN {X 0,Y 353.671,Z 394.637,A -85,B 0,C 180,E1 7731.438,E2 7731.438} C_VEL
LIN {X 0,Y 338.378,Z 577.579,A -85,B 0,C 180,E1 7727.387,E2 7727.387} C_VEL
LIN {X 0,Y 335.521,Z 598.336,A -85,B 0,C 180,E1 7726.666,E2 7726.666} C_VEL
LIN {X 0,Y 331.718,Z 618.665,A -85,B 0,C 180,E1 7725.692,E2 7725.692} C_VEL
LIN {X 0,Y 326.961,Z 638.771,A -85,B 0,C 180,E1 7724.43,E2 7724.43} C_VEL
LIN {X 0,Y 321.633,Z 657.615,A -85,B 0,C 180,E1 7722.93,E2 7722.93} C_VEL
LIN {X 0,Y 315.516,Z 676.2,A -85,B 0,C 180,E1 7721.078,E2 7721.078} C_VEL
LIN {X 0,Y 309.085,Z 693.275,A -85,B 0,C 180,E1 7718.959,E2 7718.959} C_VEL
LIN {X 0,Y 302.484,Z 709.233,A -85,B 0,C 180,E1 7716.534,E2 7716.534} C_VEL
LIN {X 0,Y 295.619,Z 724.536,A -85,B 0,C 180,E1 7713.679,E2 7713.679} C_VEL
LIN {X 0,Y 289.235,Z 737.98,A -85,B 0,C 180,E1 7710.594,E2 7710.594} C_VEL
LIN {X 0,Y 283.246,Z 750.166,A -85,B 0,C 180,E1 7707.158,E2 7707.158} C_VEL
LIN {X 0,Y 277.76,Z 761.062,A -85,B 0,C 180,E1 7703.308,E2 7703.308} C_VEL
LIN {X 0,Y 273.246,Z 770.166,A -85,B 0,C 180,E1 7699.243,E2 7699.243} C_VEL
LIN {X 0,Y 269.801,Z 777.463,A -85,B 0,C 180,E1 7695.061,E2 7695.061} C_VEL
LIN {X 0,Y 267.296,Z 783.315,A -85,B 0,C 180,E1 7690.597,E2 7690.597} C_VEL
LIN {X 0,Y 265.797,Z 787.372,A -85,B 0,C 180,E1 7686.201,E2 7686.201} C_VEL
LIN {X 0,Y 265.041,Z 789.767,A -85,B 0,C 180,E1 7681.883,E2 7681.883} C_VEL
LIN {X 0,Y 264.751,Z 790.682,A -85,B 0,C 180,E1 7677.681,E2 7677.681} C_VEL
LIN {X 0,Y 264.751,Z 790.265,A -85,B 0,C 180,E1 7673.413,E2 7673.413} C_VEL
LIN {X 0,Y 265.046,Z 788.396,A -85,B 0,C 180,E1 7669.162,E2 7669.162} C_VEL
LIN {X 0,Y 265.83,Z 784.957,A -85,B 0,C 180,E1 7664.821,E2 7664.821} C_VEL
LIN {X 0,Y 267.411,Z 779.732,A -85,B 0,C 180,E1 7660.341,E2 7660.341} C_VEL
LIN {X 0,Y 269.777,Z 773.177,A -85,B 0,C 180,E1 7656.172,E2 7656.172} C_VEL
LIN {X 0,Y 273.283,Z 764.43,A -85,B 0,C 180,E1 7651.889,E2 7651.889} C_VEL
LIN {X 0,Y 277.61,Z 754.149,A -85,B 0,C 180,E1 7647.938,E2 7647.938} C_VEL
LIN {X 0,Y 282.321,Z 743.124,A -85,B 0,C 180,E1 7644.515,E2 7644.515} C_VEL
LIN {X 0,Y 287.813,Z 730.145,A -85,B 0,C 180,E1 7641.21,E2 7641.21} C_VEL
LIN {X 0,Y 293.675,Z 715.775,A -85,B 0,C 180,E1 7638.215,E2 7638.215} C_VEL
LIN {X 0,Y 299.553,Z 700.52,A -85,B 0,C 180,E1 7635.603,E2 7635.603} C_VEL
LIN {X 0,Y 305.662,Z 683.066,A -85,B 0,C 180,E1 7633.175,E2 7633.175} C_VEL
LIN {X 0,Y 311.265,Z 665.245,A -85,B 0,C 180,E1 7631.168,E2 7631.168} C_VEL
LIN {X 0,Y 316.409,Z 646.613,A -85,B 0,C 180,E1 7629.468,E2 7629.468} C_VEL
LIN {X 0,Y 321.216,Z 625.963,A -85,B 0,C 180,E1 7627.973,E2 7627.973} C_VEL
LIN {X 0,Y 325.085,Z 605.431,A -85,B 0,C 180,E1 7626.83,E2 7626.83} C_VEL
LIN {X 0,Y 328.137,Z 584.281,A -85,B 0,C 180,E1 7625.963,E2 7625.963} C_VEL
LIN {X 0,Y 330.252,Z 562.019,A -85,B 0,C 180,E1 7625.345,E2 7625.345} C_VEL
LIN {X 0,Y 341.691,Z 394.348,A -85,B 0,C 180,E1 7621.725,E2 7621.725} C_VEL
LIN {X 0,Y 341.336,Z 391.516,A -85,B 0,C 180,E1 7621.536,E2 7621.536} C_VEL
LIN {X 0,Y 339.591,Z 388.498,A -85,B 0,C 180,E1 7621.015,E2 7621.015} C_VEL
LIN {X 0,Y 335.65,Z 385.613,A -85,B 0,C 180,E1 7619.951,E2 7619.951} C_VEL
LIN {X 0,Y 332.087,Z 382.682,A -85,B 0,C 180,E1 7618.927,E2 7618.927} C_VEL
LIN {X 0,Y 331.444,Z 381.72,A -85,B 0,C 180,E1 7618.719,E2 7618.719} C_VEL
LIN {X 0,Y 322.927,Z 367.817,A -85,B 0,C 180,E1 7615.757,E2 7615.757} C_VEL
LIN {X 0,Y 314.386,Z 354.775,A -85,B 0,C 180,E1 7612.435,E2 7612.435} C_VEL
LIN {X 0,Y 307.462,Z 345.084,A -85,B 0,C 180,E1 7609.416,E2 7609.416} C_VEL
LIN {X 0,Y 301.443,Z 336.819,A -85,B 0,C 180,E1 7606.444,E2 7606.444} C_VEL
LIN {X 0,Y 294.506,Z 327.798,A -85,B 0,C 180,E1 7602.499,E2 7602.499} C_VEL
LIN {X 0,Y 290.713,Z 322.967,A -85,B 0,C 180,E1 7599.958,E2 7599.958} C_VEL
LIN {X 0,Y 285.973,Z 317.287,A -85,B 0,C 180,E1 7596.341,E2 7596.341} C_VEL
LIN {X 0,Y 284.426,Z 315.576,A -85,B 0,C 180,E1 7594.957,E2 7594.957} C_VEL
LIN {X 0,Y 280.871,Z 311.186,A -85,B 0,C 180,E1 7591.312,E2 7591.312} C_VEL
LIN {X 0,Y 275.797,Z 305.398,A -85,B 0,C 180,E1 7582.822,E2 7582.822} C_VEL
LIN {X 0,Y 274.747,Z 304.322,A -85,B 0,C 180,E1 7578.89,E2 7578.89} C_VEL
LIN {X 0,Y 274.924,Z 304.445,A -85,B 0,C 180,E1 7572.816,E2 7572.816} C_VEL
LIN {X 0,Y 275.991,Z 305.703,A -85,B 0,C 180,E1 7569.17,E2 7569.17} C_VEL
LIN {X 0,Y 281.081,Z 311.272,A -85,B 0,C 180,E1 7561.13,E2 7561.13} C_VEL
LIN {X 0,Y 284.49,Z 315.636,A -85,B 0,C 180,E1 7557.581,E2 7557.581} C_VEL
LIN {X 0,Y 286.329,Z 317.506,A -85,B 0,C 180,E1 7555.994,E2 7555.994} C_VEL
LIN {X 0,Y 290.102,Z 322.144,A -85,B 0,C 180,E1 7553.07,E2 7553.07} C_VEL
LIN {X 0,Y 291.507,Z 323.851,A -85,B 0,C 180,E1 7552.063,E2 7552.063} C_VEL
LIN {X 0,Y 296.51,Z 330.094,A -85,B 0,C 180,E1 7548.882,E2 7548.882} C_VEL
LIN {X 0,Y 301.123,Z 336.06,A -85,B 0,C 180,E1 7546.265,E2 7546.265} C_VEL
LIN {X 0,Y 304.717,Z 340.78,A -85,B 0,C 180,E1 7544.439,E2 7544.439} C_VEL
LIN {X 0,Y 308.95,Z 346.47,A -85,B 0,C 180,E1 7542.434,E2 7542.434} C_VEL
LIN {X 0,Y 315.015,Z 354.786,A -85,B 0,C 180,E1 7539.806,E2 7539.806} C_VEL
LIN {X 0,Y 323.632,Z 367.41,A -85,B 0,C 180,E1 7536.463,E2 7536.463} C_VEL
LIN {X 0,Y 333.285,Z 382.622,A -85,B 0,C 180,E1 7533.135,E2 7533.135} C_VEL
LIN {X 0,Y 341.765,Z 397.313,A -85,B 0,C 180,E1 7530.477,E2 7530.477} C_VEL
LIN {X 0,Y 328.639,Z 597.548,A -85,B 0,C 180,E1 7526.237,E2 7526.237} C_VEL
LIN {X 0,Y 325.761,Z 619.688,A -85,B 0,C 180,E1 7525.551,E2 7525.551} C_VEL
LIN {X 0,Y 321.831,Z 641.146,A -85,B 0,C 180,E1 7524.636,E2 7524.636} C_VEL
LIN {X 0,Y 317.045,Z 662.178,A -85,B 0,C 180,E1 7523.435,E2 7523.435} C_VEL
LIN {X 0,Y 311.684,Z 682.018,A -85,B 0,C 180,E1 7521.98,E2 7521.98} C_VEL
LIN {X 0,Y 305.702,Z 700.995,A -85,B 0,C 180,E1 7520.226,E2 7520.226} C_VEL
LIN {X 0,Y 299.052,Z 719.954,A -85,B 0,C 180,E1 7518.062,E2 7518.062} C_VEL
LIN {X 0,Y 292.4,Z 737.419,A -85,B 0,C 180,E1 7515.613,E2 7515.613} C_VEL
LIN {X 0,Y 285.639,Z 753.943,A -85,B 0,C 180,E1 7512.768,E2 7512.768} C_VEL
LIN {X 0,Y 279.185,Z 768.984,A -85,B 0,C 180,E1 7509.601,E2 7509.601} C_VEL
LIN {X 0,Y 272.925,Z 783.47,A -85,B 0,C 180,E1 7505.882,E2 7505.882} C_VEL
LIN {X 0,Y 267.717,Z 795.788,A -85,B 0,C 180,E1 7502.025,E2 7502.025} C_VEL
LIN {X 0,Y 263.333,Z 806.785,A -85,B 0,C 180,E1 7497.785,E2 7497.785} C_VEL
LIN {X 0,Y 260.052,Z 816.086,A -85,B 0,C 180,E1 7493.327,E2 7493.327} C_VEL
LIN {X 0,Y 257.817,Z 824.013,A -85,B 0,C 180,E1 7488.54,E2 7488.54} C_VEL
LIN {X 0,Y 256.705,Z 829.84,A -85,B 0,C 180,E1 7483.972,E2 7483.972} C_VEL
LIN {X 0,Y 256.377,Z 833.912,A -85,B 0,C 180,E1 7479.425,E2 7479.425} C_VEL
LIN {X 0,Y 256.455,Z 836.417,A -85,B 0,C 180,E1 7475.142,E2 7475.142} C_VEL
LIN {X 0,Y 256.567,Z 837.365,A -85,B 0,C 180,E1 7471.114,E2 7471.114} C_VEL
LIN {X 0,Y 256.53,Z 837.163,A -85,B 0,C 180,E1 7467.317,E2 7467.317} C_VEL
LIN {X 0,Y 256.398,Z 835.566,A -85,B 0,C 180,E1 7463.054,E2 7463.054} C_VEL
LIN {X 0,Y 256.428,Z 832.581,A -85,B 0,C 180,E1 7458.755,E2 7458.755} C_VEL
LIN {X 0,Y 257.08,Z 827.629,A -85,B 0,C 180,E1 7453.968,E2 7453.968} C_VEL
LIN {X 0,Y 258.714,Z 820.968,A -85,B 0,C 180,E1 7449.17,E2 7449.17} C_VEL
LIN {X 0,Y 261.402,Z 812.829,A -85,B 0,C 180,E1 7444.632,E2 7444.632} C_VEL
LIN {X 0,Y 265.334,Z 802.866,A -85,B 0,C 180,E1 7440.169,E2 7440.169} C_VEL
LIN {X 0,Y 270.5,Z 791.157,A -85,B 0,C 180,E1 7435.893,E2 7435.893} C_VEL
LIN {X 0,Y 276.536,Z 778.151,A -85,B 0,C 180,E1 7432.02,E2 7432.02} C_VEL
LIN {X 0,Y 283.409,Z 763.38,A -85,B 0,C 180,E1 7428.449,E2 7428.449} C_VEL
LIN {X 0,Y 290.709,Z 747.422,A -85,B 0,C 180,E1 7425.301,E2 7425.301} C_VEL
LIN {X 0,Y 298.07,Z 730.623,A -85,B 0,C 180,E1 7422.581,E2 7422.581} C_VEL
LIN {X 0,Y 305.282,Z 713.008,A -85,B 0,C 180,E1 7420.258,E2 7420.258} C_VEL
LIN {X 0,Y 312.404,Z 693.735,A -85,B 0,C 180,E1 7418.209,E2 7418.209} C_VEL
LIN {X 0,Y 318.744,Z 674.557,A -85,B 0,C 180,E1 7416.576,E2 7416.576} C_VEL
LIN {X 0,Y 324.414,Z 654.863,A -85,B 0,C 180,E1 7415.238,E2 7415.238} C_VEL
LIN {X 0,Y 329.472,Z 633.736,A -85,B 0,C 180,E1 7414.14,E2 7414.14} C_VEL
LIN {X 0,Y 333.468,Z 612.507,A -85,B 0,C 180,E1 7413.328,E2 7413.328} C_VEL
LIN {X 0,Y 336.421,Z 589.184,A -85,B 0,C 180,E1 7412.669,E2 7412.669} C_VEL
LIN {X 0,Y 351.059,Z 399.716,A -85,B 0,C 180,E1 7408.611,E2 7408.611} C_VEL
LIN {X 0,Y 346.004,Z 389.55,A -85,B 0,C 180,E1 7406.195,E2 7406.195} C_VEL
LIN {X 0,Y 341.288,Z 380.801,A -85,B 0,C 180,E1 7403.527,E2 7403.527} C_VEL
LIN {X 0,Y 337.211,Z 373.758,A -85,B 0,C 180,E1 7400.663,E2 7400.663} C_VEL
LIN {X 0,Y 334.374,Z 369.162,A -85,B 0,C 180,E1 7398.026,E2 7398.026} C_VEL
LIN {X 0,Y 331.84,Z 364.853,A -85,B 0,C 180,E1 7394.306,E2 7394.306} C_VEL
LIN {X 0,Y 330.863,Z 363.942,A -85,B 0,C 180,E1 7390.272,E2 7390.272} C_VEL
LIN {X 0,Y 331.761,Z 364.953,A -85,B 0,C 180,E1 7386.577,E2 7386.577} C_VEL
LIN {X 0,Y 334.544,Z 369.968,A -85,B 0,C 180,E1 7382.485,E2 7382.485} C_VEL
LIN {X 0,Y 337.653,Z 375.357,A -85,B 0,C 180,E1 7379.662,E2 7379.662} C_VEL
LIN {X 0,Y 341.362,Z 382.076,A -85,B 0,C 180,E1 7377.063,E2 7377.063} C_VEL
LIN {X 0,Y 345.6,Z 389.945,A -85,B 0,C 180,E1 7374.648,E2 7374.648} C_VEL
LIN {X 0,Y 349.867,Z 398.729,A -85,B 0,C 180,E1 7372.53,E2 7372.53} C_VEL
LIN {X 0,Y 334.273,Z 577.976,A -85,B 0,C 180,E1 7368.556,E2 7368.556} C_VEL
LIN {X 0,Y 331.327,Z 598.62,A -85,B 0,C 180,E1 7367.841,E2 7367.841} C_VEL
LIN {X 0,Y 327.491,Z 618.512,A -85,B 0,C 180,E1 7366.895,E2 7366.895} C_VEL
LIN {X 0,Y 322.932,Z 637.506,A -85,B 0,C 180,E1 7365.726,E2 7365.726} C_VEL
LIN {X 0,Y 317.403,Z 656.629,A -85,B 0,C 180,E1 7364.235,E2 7364.235} C_VEL
LIN {X 0,Y 311.093,Z 675.088,A -85,B 0,C 180,E1 7362.417,E2 7362.417} C_VEL
LIN {X 0,Y 304.639,Z 691.799,A -85,B 0,C 180,E1 7360.388,E2 7360.388} C_VEL
LIN {X 0,Y 297.526,Z 708.477,A -85,B 0,C 180,E1 7357.892,E2 7357.892} C_VEL
LIN {X 0,Y 290.502,Z 723.564,A -85,B 0,C 180,E1 7355.112,E2 7355.112} C_VEL
LIN {X 0,Y 283.842,Z 737.04,A -85,B 0,C 180,E1 7352.065,E2 7352.065} C_VEL
LIN {X 0,Y 277.174,Z 749.813,A -85,B 0,C 180,E1 7348.465,E2 7348.465} C_VEL
LIN {X 0,Y 271.429,Z 760.586,A -85,B 0,C 180,E1 7344.669,E2 7344.669} C_VEL
LIN {X 0,Y 266.565,Z 769.77,A -85,B 0,C 180,E1 7340.598,E2 7340.598} C_VEL
LIN {X 0,Y 262.586,Z 777.606,A -85,B 0,C 180,E1 7336.135,E2 7336.135} C_VEL
LIN {X 0,Y 259.862,Z 783.45,A -85,B 0,C 180,E1 7331.721,E2 7331.721} C_VEL
LIN {X 0,Y 258.068,Z 787.785,A -85,B 0,C 180,E1 7327.053,E2 7327.053} C_VEL
LIN {X 0,Y 257.18,Z 790.247,A -85,B 0,C 180,E1 7322.713,E2 7322.713} C_VEL
LIN {X 0,Y 256.802,Z 791.393,A -85,B 0,C 180,E1 7318.109,E2 7318.109} C_VEL
LIN {X 0,Y 256.776,Z 791.108,A -85,B 0,C 180,E1 7313.792,E2 7313.792} C_VEL
LIN {X 0,Y 257.061,Z 789.264,A -85,B 0,C 180,E1 7309.308,E2 7309.308} C_VEL
LIN {X 0,Y 257.863,Z 785.938,A -85,B 0,C 180,E1 7304.83,E2 7304.83} C_VEL
LIN {X 0,Y 259.392,Z 781.139,A -85,B 0,C 180,E1 7300.44,E2 7300.44} C_VEL
LIN {X 0,Y 261.949,Z 774.396,A -85,B 0,C 180,E1 7295.918,E2 7295.918} C_VEL
LIN {X 0,Y 265.581,Z 765.73,A -85,B 0,C 180,E1 7291.512,E2 7291.512} C_VEL
LIN {X 0,Y 270.07,Z 755.574,A -85,B 0,C 180,E1 7287.456,E2 7287.456} C_VEL
LIN {X 0,Y 275.271,Z 744.007,A -85,B 0,C 180,E1 7283.746,E2 7283.746} C_VEL
LIN {X 0,Y 281.002,Z 731.056,A -85,B 0,C 180,E1 7280.375,E2 7280.375} C_VEL
LIN {X 0,Y 287.105,Z 716.718,A -85,B 0,C 180,E1 7277.328,E2 7277.328} C_VEL
LIN {X 0,Y 293.422,Z 700.917,A -85,B 0,C 180,E1 7274.588,E2 7274.588} C_VEL
LIN {X 0,Y 299.775,Z 683.426,A -85,B 0,C 180,E1 7272.133,E2 7272.133} C_VEL
LIN {X 0,Y 305.588,Z 665.554,A -85,B 0,C 180,E1 7270.108,E2 7270.108} C_VEL
LIN {X 0,Y 310.912,Z 646.865,A -85,B 0,C 180,E1 7268.396,E2 7268.396} C_VEL
LIN {X 0,Y 315.882,Z 626.145,A -85,B 0,C 180,E1 7266.892,E2 7266.892} C_VEL
LIN {X 0,Y 319.897,Z 605.414,A -85,B 0,C 180,E1 7265.74,E2 7265.74} C_VEL
LIN {X 0,Y 323.012,Z 584.358,A -85,B 0,C 180,E1 7264.88,E2 7264.88} C_VEL
LIN {X 0,Y 325.169,Z 562.241,A -85,B 0,C 180,E1 7264.265,E2 7264.265} C_VEL
LIN {X 0,Y 337.118,Z 391.815,A -85,B 0,C 180,E1 7260.554,E2 7260.554} C_VEL
LIN {X 0,Y 331.444,Z 381.72,A -85,B 0,C 180,E1 7258.719,E2 7258.719} C_VEL
LIN {X 0,Y 328.729,Z 378.265,A -85,B 0,C 180,E1 7257.852,E2 7257.852} C_VEL
LIN {X 0,Y 323.246,Z 374.447,A -85,B 0,C 180,E1 7256.152,E2 7256.152} C_VEL
LIN {X 0,Y 317.947,Z 370.711,A -85,B 0,C 180,E1 7254.384,E2 7254.384} C_VEL
LIN {X 0,Y 315.852,Z 368.012,A -85,B 0,C 180,E1 7253.584,E2 7253.584} C_VEL
LIN {X 0,Y 308.803,Z 357.521,A -85,B 0,C 180,E1 7250.611,E2 7250.611} C_VEL
LIN {X 0,Y 302.546,Z 348.657,A -85,B 0,C 180,E1 7247.657,E2 7247.657} C_VEL
LIN {X 0,Y 296.695,Z 340.531,A -85,B 0,C 180,E1 7244.501,E2 7244.501} C_VEL
LIN {X 0,Y 292.147,Z 334.765,A -85,B 0,C 180,E1 7241.751,E2 7241.751} C_VEL
LIN {X 0,Y 288.09,Z 329.507,A -85,B 0,C 180,E1 7238.914,E2 7238.914} C_VEL
LIN {X 0,Y 284.295,Z 324.703,A -85,B 0,C 180,E1 7235.841,E2 7235.841} C_VEL
LIN {X 0,Y 279.604,Z 319.101,A -85,B 0,C 180,E1 7231.111,E2 7231.111} C_VEL
LIN {X 0,Y 274.978,Z 313.811,A -85,B 0,C 180,E1 7223.574,E2 7223.574} C_VEL
LIN {X 0,Y 273.851,Z 312.366,A -85,B 0,C 180,E1 7219.847,E2 7219.847} C_VEL
LIN {X 0,Y 273.734,Z 312.263,A -85,B 0,C 180,E1 7213.517,E2 7213.517} C_VEL
LIN {X 0,Y 274.79,Z 313.427,A -85,B 0,C 180,E1 7209.592,E2 7209.592} C_VEL
LIN {X 0,Y 279.729,Z 319.033,A -85,B 0,C 180,E1 7201.432,E2 7201.432} C_VEL
LIN {X 0,Y 283.196,Z 323.483,A -85,B 0,C 180,E1 7197.773,E2 7197.773} C_VEL
LIN {X 0,Y 284.767,Z 325.143,A -85,B 0,C 180,E1 7196.375,E2 7196.375} C_VEL
LIN {X 0,Y 288.749,Z 330.013,A -85,B 0,C 180,E1 7193.237,E2 7193.237} C_VEL
LIN {X 0,Y 294.575,Z 337.496,A -85,B 0,C 180,E1 7189.338,E2 7189.338} C_VEL
LIN {X 0,Y 301.154,Z 345.975,A -85,B 0,C 180,E1 7185.629,E2 7185.629} C_VEL
LIN {X 0,Y 309.188,Z 357.106,A -85,B 0,C 180,E1 7181.766,E2 7181.766} C_VEL
LIN {X 0,Y 317.72,Z 369.526,A -85,B 0,C 180,E1 7178.2,E2 7178.2} C_VEL
LIN {X 0,Y 326.599,Z 383.463,A -85,B 0,C 180,E1 7174.911,E2 7174.911} C_VEL
LIN {X 0,Y 335.84,Z 399.056,A -85,B 0,C 180,E1 7171.842,E2 7171.842} C_VEL
LIN {X 0,Y 336.874,Z 401.296,A -85,B 0,C 180,E1 7171.5,E2 7171.5} C_VEL
LIN {X 0,Y 323.57,Z 597.173,A -85,B 0,C 180,E1 7167.332,E2 7167.332} C_VEL
LIN {X 0,Y 320.615,Z 619.347,A -85,B 0,C 180,E1 7166.644,E2 7166.644} C_VEL
LIN {X 0,Y 316.79,Z 639.785,A -85,B 0,C 180,E1 7165.78,E2 7165.78} C_VEL
LIN {X 0,Y 312.051,Z 660.344,A -85,B 0,C 180,E1 7164.628,E2 7164.628} C_VEL
LIN {X 0,Y 306.571,Z 680.123,A -85,B 0,C 180,E1 7163.191,E2 7163.191} C_VEL
LIN {X 0,Y 300.435,Z 699.203,A -85,B 0,C 180,E1 7161.448,E2 7161.448} C_VEL
LIN {X 0,Y 293.537,Z 718.377,A -85,B 0,C 180,E1 7159.274,E2 7159.274} C_VEL
LIN {X 0,Y 286.6,Z 736.005,A -85,B 0,C 180,E1 7156.81,E2 7156.81} C_VEL
LIN {X 0,Y 279.531,Z 752.63,A -85,B 0,C 180,E1 7153.938,E2 7153.938} C_VEL
LIN {X 0,Y 272.774,Z 767.817,A -85,B 0,C 180,E1 7150.724,E2 7150.724} C_VEL
LIN {X 0,Y 266.163,Z 782.39,A -85,B 0,C 180,E1 7146.942,E2 7146.942} C_VEL
LIN {X 0,Y 260.646,Z 794.783,A -85,B 0,C 180,E1 7143.003,E2 7143.003} C_VEL
LIN {X 0,Y 256.014,Z 805.711,A -85,B 0,C 180,E1 7138.707,E2 7138.707} C_VEL
LIN {X 0,Y 252.431,Z 815.201,A -85,B 0,C 180,E1 7134.075,E2 7134.075} C_VEL
LIN {X 0,Y 250.067,Z 822.921,A -85,B 0,C 180,E1 7129.329,E2 7129.329} C_VEL
LIN {X 0,Y 248.82,Z 828.759,A -85,B 0,C 180,E1 7124.662,E2 7124.662} C_VEL
LIN {X 0,Y 248.404,Z 832.972,A -85,B 0,C 180,E1 7119.964,E2 7119.964} C_VEL
LIN {X 0,Y 248.463,Z 835.581,A -85,B 0,C 180,E1 7115.54,E2 7115.54} C_VEL
LIN {X 0,Y 248.594,Z 836.624,A -85,B 0,C 180,E1 7111.38,E2 7111.38} C_VEL
LIN {X 0,Y 248.572,Z 836.517,A -85,B 0,C 180,E1 7107.692,E2 7107.692} C_VEL
LIN {X 0,Y 248.426,Z 835.126,A -85,B 0,C 180,E1 7103.295,E2 7103.295} C_VEL
LIN {X 0,Y 248.434,Z 832.242,A -85,B 0,C 180,E1 7098.859,E2 7098.859} C_VEL
LIN {X 0,Y 249.083,Z 827.497,A -85,B 0,C 180,E1 7093.918,E2 7093.918} C_VEL
LIN {X 0,Y 250.658,Z 821.347,A -85,B 0,C 180,E1 7089.203,E2 7089.203} C_VEL
LIN {X 0,Y 253.383,Z 813.464,A -85,B 0,C 180,E1 7084.523,E2 7084.523} C_VEL
LIN {X 0,Y 257.639,Z 803.325,A -85,B 0,C 180,E1 7079.699,E2 7079.699} C_VEL
LIN {X 0,Y 262.795,Z 792.31,A -85,B 0,C 180,E1 7075.463,E2 7075.463} C_VEL
LIN {X 0,Y 269.186,Z 779.185,A -85,B 0,C 180,E1 7071.388,E2 7071.388} C_VEL
LIN {X 0,Y 276.373,Z 764.588,A -85,B 0,C 180,E1 7067.706,E2 7067.706} C_VEL
LIN {X 0,Y 283.989,Z 748.902,A -85,B 0,C 180,E1 7064.479,E2 7064.479} C_VEL
LIN {X 0,Y 291.77,Z 732.074,A -85,B 0,C 180,E1 7061.661,E2 7061.661} C_VEL
LIN {X 0,Y 299.482,Z 714.051,A -85,B 0,C 180,E1 7059.232,E2 7059.232} C_VEL
LIN {X 0,Y 306.695,Z 695.52,A -85,B 0,C 180,E1 7057.213,E2 7057.213} C_VEL
LIN {X 0,Y 313.735,Z 675.297,A -85,B 0,C 180,E1 7055.453,E2 7055.453} C_VEL
LIN {X 0,Y 319.847,Z 655.026,A -85,B 0,C 180,E1 7054.063,E2 7054.063} C_VEL
LIN {X 0,Y 325.046,Z 634.075,A -85,B 0,C 180,E1 7052.974,E2 7052.974} C_VEL
LIN {X 0,Y 329.243,Z 612.681,A -85,B 0,C 180,E1 7052.152,E2 7052.152} C_VEL
LIN {X 0,Y 332.325,Z 589.646,A -85,B 0,C 180,E1 7051.494,E2 7051.494} C_VEL
LIN {X 0,Y 347.339,Z 403.954,A -85,B 0,C 180,E1 7047.501,E2 7047.501} C_VEL
LIN {X 0,Y 342.525,Z 394.166,A -85,B 0,C 180,E1 7044.996,E2 7044.996} C_VEL
LIN {X 0,Y 338.38,Z 386.393,A -85,B 0,C 180,E1 7042.408,E2 7042.408} C_VEL
LIN {X 0,Y 335.246,Z 380.764,A -85,B 0,C 180,E1 7039.969,E2 7039.969} C_VEL
LIN {X 0,Y 332.937,Z 376.789,A -85,B 0,C 180,E1 7037.658,E2 7037.658} C_VEL
LIN {X 0,Y 330.705,Z 372.739,A -85,B 0,C 180,E1 7034.177,E2 7034.177} C_VEL
LIN {X 0,Y 329.793,Z 371.87,A -85,B 0,C 180,E1 7030.306,E2 7030.306} C_VEL
LIN {X 0,Y 330.583,Z 372.8,A -85,B 0,C 180,E1 7026.776,E2 7026.776} C_VEL
LIN {X 0,Y 333.159,Z 377.726,A -85,B 0,C 180,E1 7022.754,E2 7022.754} C_VEL
LIN {X 0,Y 336.059,Z 382.957,A -85,B 0,C 180,E1 7020.001,E2 7020.001} C_VEL
LIN {X 0,Y 339.502,Z 389.507,A -85,B 0,C 180,E1 7017.47,E2 7017.47} C_VEL
LIN {X 0,Y 343.409,Z 397.186,A -85,B 0,C 180,E1 7015.116,E2 7015.116} C_VEL
LIN {X 0,Y 346.176,Z 403.286,A -85,B 0,C 180,E1 7013.638,E2 7013.638} C_VEL
LIN {X 0,Y 330.326,Z 578.552,A -85,B 0,C 180,E1 7009.751,E2 7009.751} C_VEL
LIN {X 0,Y 327.249,Z 599.421,A -85,B 0,C 180,E1 7009.03,E2 7009.03} C_VEL
LIN {X 0,Y 323.355,Z 618.935,A -85,B 0,C 180,E1 7008.105,E2 7008.105} C_VEL
LIN {X 0,Y 318.643,Z 637.87,A -85,B 0,C 180,E1 7006.944,E2 7006.944} C_VEL
LIN {X 0,Y 312.968,Z 656.772,A -85,B 0,C 180,E1 7005.474,E2 7005.474} C_VEL
LIN {X 0,Y 306.62,Z 674.781,A -85,B 0,C 180,E1 7003.716,E2 7003.716} C_VEL
LIN {X 0,Y 299.729,Z 691.999,A -85,B 0,C 180,E1 7001.637,E2 7001.637} C_VEL
LIN {X 0,Y 292.199,Z 708.935,A -85,B 0,C 180,E1 6999.097,E2 6999.097} C_VEL
LIN {X 0,Y 284.941,Z 723.893,A -85,B 0,C 180,E1 6996.331,E2 6996.331} C_VEL
LIN {X 0,Y 277.811,Z 737.587,A -85,B 0,C 180,E1 6993.201,E2 6993.201} C_VEL
LIN {X 0,Y 270.924,Z 750.121,A -85,B 0,C 180,E1 6989.631,E2 6989.631} C_VEL
LIN {X 0,Y 264.802,Z 760.952,A -85,B 0,C 180,E1 6985.767,E2 6985.767} C_VEL
LIN {X 0,Y 259.445,Z 770.462,A -85,B 0,C 180,E1 6981.477,E2 6981.477} C_VEL
LIN {X 0,Y 255.288,Z 778.089,A -85,B 0,C 180,E1 6977.043,E2 6977.043} C_VEL
LIN {X 0,Y 252.227,Z 784.133,A -85,B 0,C 180,E1 6972.371,E2 6972.371} C_VEL
LIN {X 0,Y 250.212,Z 788.6,A -85,B 0,C 180,E1 6967.404,E2 6967.404} C_VEL
LIN {X 0,Y 249.231,Z 791.073,A -85,B 0,C 180,E1 6962.794,E2 6962.794} C_VEL
LIN {X 0,Y 248.832,Z 792.127,A -85,B 0,C 180,E1 6958.045,E2 6958.045} C_VEL
LIN {X 0,Y 248.811,Z 791.783,A -85,B 0,C 180,E1 6953.626,E2 6953.626} C_VEL
LIN {X 0,Y 249.105,Z 790.006,A -85,B 0,C 180,E1 6949.218,E2 6949.218} C_VEL
LIN {X 0,Y 249.968,Z 786.653,A -85,B 0,C 180,E1 6944.548,E2 6944.548} C_VEL
LIN {X 0,Y 251.674,Z 781.65,A -85,B 0,C 180,E1 6939.865,E2 6939.865} C_VEL
LIN {X 0,Y 254.282,Z 775.197,A -85,B 0,C 180,E1 6935.417,E2 6935.417} C_VEL
LIN {X 0,Y 258.11,Z 766.542,A -85,B 0,C 180,E1 6930.89,E2 6930.89} C_VEL
LIN {X 0,Y 262.825,Z 756.406,A -85,B 0,C 180,E1 6926.731,E2 6926.731} C_VEL
LIN {X 0,Y 268.268,Z 744.864,A -85,B 0,C 180,E1 6922.937,E2 6922.937} C_VEL
LIN {X 0,Y 274.625,Z 731.112,A -85,B 0,C 180,E1 6919.301,E2 6919.301} C_VEL
LIN {X 0,Y 281.076,Z 716.527,A -85,B 0,C 180,E1 6916.188,E2 6916.188} C_VEL
LIN {X 0,Y 287.613,Z 700.716,A -85,B 0,C 180,E1 6913.44,E2 6913.44} C_VEL
LIN {X 0,Y 294.24,Z 683.104,A -85,B 0,C 180,E1 6910.963,E2 6910.963} C_VEL
LIN {X 0,Y 300.54,Z 664.241,A -85,B 0,C 180,E1 6908.843,E2 6908.843} C_VEL
LIN {X 0,Y 306.059,Z 645.109,A -85,B 0,C 180,E1 6907.125,E2 6907.125} C_VEL
LIN {X 0,Y 310.654,Z 626.234,A -85,B 0,C 180,E1 6905.775,E2 6905.775} C_VEL
LIN {X 0,Y 314.843,Z 605.091,A -85,B 0,C 180,E1 6904.607,E2 6904.607} C_VEL
LIN {X 0,Y 318.007,Z 584.056,A -85,B 0,C 180,E1 6903.755,E2 6903.755} C_VEL
LIN {X 0,Y 320.2,Z 561.992,A -85,B 0,C 180,E1 6903.146,E2 6903.146} C_VEL
LIN {X 0,Y 332.286,Z 395.58,A -85,B 0,C 180,E1 6899.504,E2 6899.504} C_VEL
LIN {X 0,Y 324.062,Z 381.206,A -85,B 0,C 180,E1 6896.69,E2 6896.69} C_VEL
LIN {X 0,Y 315.852,Z 368.012,A -85,B 0,C 180,E1 6893.584,E2 6893.584} C_VEL
LIN {X 0,Y 313.339,Z 365.06,A -85,B 0,C 180,E1 6892.601,E2 6892.601} C_VEL
LIN {X 0,Y 308.562,Z 362.509,A -85,B 0,C 180,E1 6890.795,E2 6890.795} C_VEL
LIN {X 0,Y 303.535,Z 359.878,A -85,B 0,C 180,E1 6888.728,E2 6888.728} C_VEL
LIN {X 0,Y 301.647,Z 357.638,A -85,B 0,C 180,E1 6887.825,E2 6887.825} C_VEL
LIN {X 0,Y 294.609,Z 347.814,A -85,B 0,C 180,E1 6883.991,E2 6883.991} C_VEL
LIN {X 0,Y 290.268,Z 342.185,A -85,B 0,C 180,E1 6881.283,E2 6881.283} C_VEL
LIN {X 0,Y 286.298,Z 336.981,A -85,B 0,C 180,E1 6878.433,E2 6878.433} C_VEL
LIN {X 0,Y 282.569,Z 332.016,A -85,B 0,C 180,E1 6875.283,E2 6875.283} C_VEL
LIN {X 0,Y 278.425,Z 327.165,A -85,B 0,C 180,E1 6871.017,E2 6871.017} C_VEL
LIN {X 0,Y 277.433,Z 325.897,A -85,B 0,C 180,E1 6869.714,E2 6869.714} C_VEL
LIN {X 0,Y 273.343,Z 320.898,A -85,B 0,C 180,E1 6861.905,E2 6861.905} C_VEL
LIN {X 0,Y 272.524,Z 320.1,A -85,B 0,C 180,E1 6857.286,E2 6857.286} C_VEL
LIN {X 0,Y 273.132,Z 320.587,A -85,B 0,C 180,E1 6851.613,E2 6851.613} C_VEL
LIN {X 0,Y 274.263,Z 322.314,A -85,B 0,C 180,E1 6848.172,E2 6848.172} C_VEL
LIN {X 0,Y 278.458,Z 326.927,A -85,B 0,C 180,E1 6841.644,E2 6841.644} C_VEL
LIN {X 0,Y 282.011,Z 331.432,A -85,B 0,C 180,E1 6837.865,E2 6837.865} C_VEL
LIN {X 0,Y 283.324,Z 332.962,A -85,B 0,C 180,E1 6836.66,E2 6836.66} C_VEL
LIN {X 0,Y 288.093,Z 338.989,A -85,B 0,C 180,E1 6832.871,E2 6832.871} C_VEL
LIN {X 0,Y 292.784,Z 345.082,A -85,B 0,C 180,E1 6829.72,E2 6829.72} C_VEL
LIN {X 0,Y 299.018,Z 353.286,A -85,B 0,C 180,E1 6826.117,E2 6826.117} C_VEL
LIN {X 0,Y 306.723,Z 364.166,A -85,B 0,C 180,E1 6822.302,E2 6822.302} C_VEL
LIN {X 0,Y 314.915,Z 376.318,A -85,B 0,C 180,E1 6818.779,E2 6818.779} C_VEL
LIN {X 0,Y 323.559,Z 390.108,A -85,B 0,C 180,E1 6815.488,E2 6815.488} C_VEL
LIN {X 0,Y 332.094,Z 404.771,A -85,B 0,C 180,E1 6812.564,E2 6812.564} C_VEL
LIN {X 0,Y 318.597,Z 596.806,A -85,B 0,C 180,E1 6808.457,E2 6808.457} C_VEL
LIN {X 0,Y 315.574,Z 618.91,A -85,B 0,C 180,E1 6807.77,E2 6807.77} C_VEL
LIN {X 0,Y 311.548,Z 639.79,A -85,B 0,C 180,E1 6806.887,E2 6806.887} C_VEL
LIN {X 0,Y 306.678,Z 660.227,A -85,B 0,C 180,E1 6805.735,E2 6805.735} C_VEL
LIN {X 0,Y 301.041,Z 679.981,A -85,B 0,C 180,E1 6804.294,E2 6804.294} C_VEL
LIN {X 0,Y 294.719,Z 699.025,A -85,B 0,C 180,E1 6802.544,E2 6802.544} C_VEL
LIN {X 0,Y 287.603,Z 718.171,A -85,B 0,C 180,E1 6800.354,E2 6800.354} C_VEL
LIN {X 0,Y 280.627,Z 735.276,A -85,B 0,C 180,E1 6797.944,E2 6797.944} C_VEL
LIN {X 0,Y 273.423,Z 751.554,A -85,B 0,C 180,E1 6795.107,E2 6795.107} C_VEL
LIN {X 0,Y 266.465,Z 766.588,A -85,B 0,C 180,E1 6791.902,E2 6791.902} C_VEL
LIN {X 0,Y 259.849,Z 780.549,A -85,B 0,C 180,E1 6788.276,E2 6788.276} C_VEL
LIN {X 0,Y 253.87,Z 793.312,A -85,B 0,C 180,E1 6784.198,E2 6784.198} C_VEL
LIN {X 0,Y 248.873,Z 804.363,A -85,B 0,C 180,E1 6779.795,E2 6779.795} C_VEL
LIN {X 0,Y 244.956,Z 814.025,A -85,B 0,C 180,E1 6775.018,E2 6775.018} C_VEL
LIN {X 0,Y 242.405,Z 821.683,A -85,B 0,C 180,E1 6770.269,E2 6770.269} C_VEL
LIN {X 0,Y 240.953,Z 827.674,A -85,B 0,C 180,E1 6765.398,E2 6765.398} C_VEL
LIN {X 0,Y 240.44,Z 832.03,A -85,B 0,C 180,E1 6760.54,E2 6760.54} C_VEL
LIN {X 0,Y 240.467,Z 834.594,A -85,B 0,C 180,E1 6756.204,E2 6756.204} C_VEL
LIN {X 0,Y 240.613,Z 835.863,A -85,B 0,C 180,E1 6751.903,E2 6751.903} C_VEL
LIN {X 0,Y 240.614,Z 835.868,A -85,B 0,C 180,E1 6748.092,E2 6748.092} C_VEL
LIN {X 0,Y 240.465,Z 834.808,A -85,B 0,C 180,E1 6744.031,E2 6744.031} C_VEL
LIN {X 0,Y 240.432,Z 832.093,A -85,B 0,C 180,E1 6739.212,E2 6739.212} C_VEL
LIN {X 0,Y 240.979,Z 827.875,A -85,B 0,C 180,E1 6734.352,E2 6734.352} C_VEL
LIN {X 0,Y 242.55,Z 821.819,A -85,B 0,C 180,E1 6729.354,E2 6729.354} C_VEL
LIN {X 0,Y 245.553,Z 813.649,A -85,B 0,C 180,E1 6724.145,E2 6724.145} C_VEL
LIN {X 0,Y 249.757,Z 804.245,A -85,B 0,C 180,E1 6719.399,E2 6719.399} C_VEL
LIN {X 0,Y 255.316,Z 792.929,A -85,B 0,C 180,E1 6714.851,E2 6714.851} C_VEL
LIN {X 0,Y 261.945,Z 780.082,A -85,B 0,C 180,E1 6710.679,E2 6710.679} C_VEL
LIN {X 0,Y 269.393,Z 765.855,A -85,B 0,C 180,E1 6706.925,E2 6706.925} C_VEL
LIN {X 0,Y 277.213,Z 750.62,A -85,B 0,C 180,E1 6703.662,E2 6703.662} C_VEL
LIN {X 0,Y 285.266,Z 734.01,A -85,B 0,C 180,E1 6700.79,E2 6700.79} C_VEL
LIN {X 0,Y 293.199,Z 716.475,A -85,B 0,C 180,E1 6698.338,E2 6698.338} C_VEL
LIN {X 0,Y 300.635,Z 698.591,A -85,B 0,C 180,E1 6696.3,E2 6696.3} C_VEL
LIN {X 0,Y 307.781,Z 679.319,A -85,B 0,C 180,E1 6694.546,E2 6694.546} C_VEL
LIN {X 0,Y 314.047,Z 659.697,A -85,B 0,C 180,E1 6693.138,E2 6693.138} C_VEL
LIN {X 0,Y 319.901,Z 638.105,A -85,B 0,C 180,E1 6691.94,E2 6691.94} C_VEL
LIN {X 0,Y 324.55,Z 616.746,A -85,B 0,C 180,E1 6691.067,E2 6691.067} C_VEL
LIN {X 0,Y 328.016,Z 594.18,A -85,B 0,C 180,E1 6690.383,E2 6690.383} C_VEL
LIN {X 0,Y 340.425,Z 446.774,A -85,B 0,C 180,E1 6687.195,E2 6687.195} C_VEL
LIN {X 0,Y 343.726,Z 408.304,A -85,B 0,C 180,E1 6686.344,E2 6686.344} C_VEL
LIN {X 0,Y 339.65,Z 399.709,A -85,B 0,C 180,E1 6684.016,E2 6684.016} C_VEL
LIN {X 0,Y 335.888,Z 392.333,A -85,B 0,C 180,E1 6681.433,E2 6681.433} C_VEL
LIN {X 0,Y 333.333,Z 387.747,A -85,B 0,C 180,E1 6679.267,E2 6679.267} C_VEL
LIN {X 0,Y 331.587,Z 384.506,A -85,B 0,C 180,E1 6677.37,E2 6677.37} C_VEL
LIN {X 0,Y 329.493,Z 380.547,A -85,B 0,C 180,E1 6673.872,E2 6673.872} C_VEL
LIN {X 0,Y 328.724,Z 379.802,A -85,B 0,C 180,E1 6670.162,E2 6670.162} C_VEL
LIN {X 0,Y 329.438,Z 380.759,A -85,B 0,C 180,E1 6666.887,E2 6666.887} C_VEL
LIN {X 0,Y 331.72,Z 385.319,A -85,B 0,C 180,E1 6663.111,E2 6663.111} C_VEL
LIN {X 0,Y 334.578,Z 390.743,A -85,B 0,C 180,E1 6660.258,E2 6660.258} C_VEL
LIN {X 0,Y 337.791,Z 397.179,A -85,B 0,C 180,E1 6657.796,E2 6657.796} C_VEL
LIN {X 0,Y 341.488,Z 404.904,A -85,B 0,C 180,E1 6655.467,E2 6655.467} C_VEL
LIN {X 0,Y 342.674,Z 407.811,A -85,B 0,C 180,E1 6654.774,E2 6654.774} C_VEL
LIN {X 0,Y 326.601,Z 579.177,A -85,B 0,C 180,E1 6650.982,E2 6650.982} C_VEL
LIN {X 0,Y 323.424,Z 599.907,A -85,B 0,C 180,E1 6650.267,E2 6650.267} C_VEL
LIN {X 0,Y 319.269,Z 619.922,A -85,B 0,C 180,E1 6649.319,E2 6649.319} C_VEL
LIN {X 0,Y 313.928,Z 640.289,A -85,B 0,C 180,E1 6648.054,E2 6648.054} C_VEL
LIN {X 0,Y 308.306,Z 658.268,A -85,B 0,C 180,E1 6646.641,E2 6646.641} C_VEL
LIN {X 0,Y 301.479,Z 676.755,A -85,B 0,C 180,E1 6644.813,E2 6644.813} C_VEL
LIN {X 0,Y 294.269,Z 693.87,A -85,B 0,C 180,E1 6642.707,E2 6642.707} C_VEL
LIN {X 0,Y 286.479,Z 710.565,A -85,B 0,C 180,E1 6640.157,E2 6640.157} C_VEL
LIN {X 0,Y 278.64,Z 725.839,A -85,B 0,C 180,E1 6637.255,E2 6637.255} C_VEL
LIN {X 0,Y 271.251,Z 739.334,A -85,B 0,C 180,E1 6634.084,E2 6634.084} C_VEL
LIN {X 0,Y 264.194,Z 751.511,A -85,B 0,C 180,E1 6630.514,E2 6630.514} C_VEL
LIN {X 0,Y 257.715,Z 762.316,A -85,B 0,C 180,E1 6626.529,E2 6626.529} C_VEL
LIN {X 0,Y 252.076,Z 771.698,A -85,B 0,C 180,E1 6622.126,E2 6622.126} C_VEL
LIN {X 0,Y 247.498,Z 779.532,A -85,B 0,C 180,E1 6617.332,E2 6617.332} C_VEL
LIN {X 0,Y 244.304,Z 785.399,A -85,B 0,C 180,E1 6612.479,E2 6612.479} C_VEL
LIN {X 0,Y 242.311,Z 789.52,A -85,B 0,C 180,E1 6607.608,E2 6607.608} C_VEL
LIN {X 0,Y 241.259,Z 791.961,A -85,B 0,C 180,E1 6602.727,E2 6602.727} C_VEL
LIN {X 0,Y 240.863,Z 792.864,A -85,B 0,C 180,E1 6597.977,E2 6597.977} C_VEL
LIN {X 0,Y 240.847,Z 792.445,A -85,B 0,C 180,E1 6593.449,E2 6593.449} C_VEL
LIN {X 0,Y 241.182,Z 790.619,A -85,B 0,C 180,E1 6588.869,E2 6588.869} C_VEL
LIN {X 0,Y 242.147,Z 787.147,A -85,B 0,C 180,E1 6584,E2 6584} C_VEL
LIN {X 0,Y 244.129,Z 781.765,A -85,B 0,C 180,E1 6578.956,E2 6578.956} C_VEL
LIN {X 0,Y 246.982,Z 775.181,A -85,B 0,C 180,E1 6574.414,E2 6574.414} C_VEL
LIN {X 0,Y 251.143,Z 766.402,A -85,B 0,C 180,E1 6569.774,E2 6569.774} C_VEL
LIN {X 0,Y 256.212,Z 756.083,A -85,B 0,C 180,E1 6565.526,E2 6565.526} C_VEL
LIN {X 0,Y 261.667,Z 745.019,A -85,B 0,C 180,E1 6561.875,E2 6561.875} C_VEL
LIN {X 0,Y 267.955,Z 731.99,A -85,B 0,C 180,E1 6558.378,E2 6558.378} C_VEL
LIN {X 0,Y 274.613,Z 717.556,A -85,B 0,C 180,E1 6555.237,E2 6555.237} C_VEL
LIN {X 0,Y 281.217,Z 702.245,A -85,B 0,C 180,E1 6552.519,E2 6552.519} C_VEL
LIN {X 0,Y 288.053,Z 684.73,A -85,B 0,C 180,E1 6550.01,E2 6550.01} C_VEL
LIN {X 0,Y 294.283,Z 666.859,A -85,B 0,C 180,E1 6547.951,E2 6547.951} C_VEL
LIN {X 0,Y 299.968,Z 648.194,A -85,B 0,C 180,E1 6546.217,E2 6546.217} C_VEL
LIN {X 0,Y 305.146,Z 628.053,A -85,B 0,C 180,E1 6544.731,E2 6544.731} C_VEL
LIN {X 0,Y 309.412,Z 607.632,A -85,B 0,C 180,E1 6543.57,E2 6543.57} C_VEL
LIN {X 0,Y 312.845,Z 586.137,A -85,B 0,C 180,E1 6542.671,E2 6542.671} C_VEL
LIN {X 0,Y 315.221,Z 563.563,A -85,B 0,C 180,E1 6542.033,E2 6542.033} C_VEL
LIN {X 0,Y 327.578,Z 399.523,A -85,B 0,C 180,E1 6538.445,E2 6538.445} C_VEL
LIN {X 0,Y 319.818,Z 385.805,A -85,B 0,C 180,E1 6535.66,E2 6535.66} C_VEL
LIN {X 0,Y 311.868,Z 372.958,A -85,B 0,C 180,E1 6532.509,E2 6532.509} C_VEL
LIN {X 0,Y 304.444,Z 361.69,A -85,B 0,C 180,E1 6529.193,E2 6529.193} C_VEL
LIN {X 0,Y 301.647,Z 357.638,A -85,B 0,C 180,E1 6527.825,E2 6527.825} C_VEL
LIN {X 0,Y 299.434,Z 355.229,A -85,B 0,C 180,E1 6526.724,E2 6526.724} C_VEL
LIN {X 0,Y 295.5,Z 353.805,A -85,B 0,C 180,E1 6524.841,E2 6524.841} C_VEL
LIN {X 0,Y 291.167,Z 352.539,A -85,B 0,C 180,E1 6522.577,E2 6522.577} C_VEL
LIN {X 0,Y 289.39,Z 350.734,A -85,B 0,C 180,E1 6521.467,E2 6521.467} C_VEL
LIN {X 0,Y 284.524,Z 344.447,A -85,B 0,C 180,E1 6517.947,E2 6517.947} C_VEL
LIN {X 0,Y 280.505,Z 339.115,A -85,B 0,C 180,E1 6514.398,E2 6514.398} C_VEL
LIN {X 0,Y 276.924,Z 334.61,A -85,B 0,C 180,E1 6510.481,E2 6510.481} C_VEL
LIN {X 0,Y 272.38,Z 328.994,A -85,B 0,C 180,E1 6502.213,E2 6502.213} C_VEL
LIN {X 0,Y 271.515,Z 328.067,A -85,B 0,C 180,E1 6498.188,E2 6498.188} C_VEL
LIN {X 0,Y 271.89,Z 328.354,A -85,B 0,C 180,E1 6492.313,E2 6492.313} C_VEL
LIN {X 0,Y 272.852,Z 329.717,A -85,B 0,C 180,E1 6489.064,E2 6489.064} C_VEL
LIN {X 0,Y 277.19,Z 334.823,A -85,B 0,C 180,E1 6481.859,E2 6481.859} C_VEL
LIN {X 0,Y 280.828,Z 339.379,A -85,B 0,C 180,E1 6477.958,E2 6477.958} C_VEL
LIN {X 0,Y 282.211,Z 341.293,A -85,B 0,C 180,E1 6476.647,E2 6476.647} C_VEL
LIN {X 0,Y 286.334,Z 346.452,A -85,B 0,C 180,E1 6473.331,E2 6473.331} C_VEL
LIN {X 0,Y 291,Z 352.667,A -85,B 0,C 180,E1 6470.106,E2 6470.106} C_VEL
LIN {X 0,Y 296.904,Z 360.594,A -85,B 0,C 180,E1 6466.612,E2 6466.612} C_VEL
LIN {X 0,Y 304.378,Z 371.368,A -85,B 0,C 180,E1 6462.803,E2 6462.803} C_VEL
LIN {X 0,Y 312.143,Z 383.108,A -85,B 0,C 180,E1 6459.367,E2 6459.367} C_VEL
LIN {X 0,Y 320.538,Z 396.747,A -85,B 0,C 180,E1 6456.076,E2 6456.076} C_VEL
LIN {X 0,Y 327.377,Z 408.714,A -85,B 0,C 180,E1 6453.639,E2 6453.639} C_VEL
LIN {X 0,Y 313.73,Z 596.502,A -85,B 0,C 180,E1 6449.614,E2 6449.614} C_VEL
LIN {X 0,Y 310.62,Z 618.669,A -85,B 0,C 180,E1 6448.924,E2 6448.924} C_VEL
LIN {X 0,Y 306.427,Z 639.789,A -85,B 0,C 180,E1 6448.03,E2 6448.03} C_VEL
LIN {X 0,Y 301.423,Z 660.109,A -85,B 0,C 180,E1 6446.88,E2 6446.88} C_VEL
LIN {X 0,Y 295.626,Z 679.814,A -85,B 0,C 180,E1 6445.438,E2 6445.438} C_VEL
LIN {X 0,Y 289.113,Z 698.786,A -85,B 0,C 180,E1 6443.683,E2 6443.683} C_VEL
LIN {X 0,Y 281.77,Z 717.877,A -85,B 0,C 180,E1 6441.48,E2 6441.48} C_VEL
LIN {X 0,Y 274.484,Z 735.098,A -85,B 0,C 180,E1 6439.027,E2 6439.027} C_VEL
LIN {X 0,Y 267,Z 751.412,A -85,B 0,C 180,E1 6436.147,E2 6436.147} C_VEL
LIN {X 0,Y 259.834,Z 766.24,A -85,B 0,C 180,E1 6432.927,E2 6432.927} C_VEL
LIN {X 0,Y 252.866,Z 780.279,A -85,B 0,C 180,E1 6429.193,E2 6429.193} C_VEL
LIN {X 0,Y 246.594,Z 793.029,A -85,B 0,C 180,E1 6425.009,E2 6425.009} C_VEL
LIN {X 0,Y 241.236,Z 804.296,A -85,B 0,C 180,E1 6420.372,E2 6420.372} C_VEL
LIN {X 0,Y 237.158,Z 813.808,A -85,B 0,C 180,E1 6415.467,E2 6415.467} C_VEL
LIN {X 0,Y 234.449,Z 821.474,A -85,B 0,C 180,E1 6410.466,E2 6410.466} C_VEL
LIN {X 0,Y 232.958,Z 827.384,A -85,B 0,C 180,E1 6405.43,E2 6405.43} C_VEL
LIN {X 0,Y 232.453,Z 831.59,A -85,B 0,C 180,E1 6400.405,E2 6400.405} C_VEL
LIN {X 0,Y 232.51,Z 834.188,A -85,B 0,C 180,E1 6395.674,E2 6395.674} C_VEL
LIN {X 0,Y 232.661,Z 835.196,A -85,B 0,C 180,E1 6391.229,E2 6391.229} C_VEL
LIN {X 0,Y 232.62,Z 835.054,A -85,B 0,C 180,E1 6387.287,E2 6387.287} C_VEL
LIN {X 0,Y 232.445,Z 833.73,A -85,B 0,C 180,E1 6382.832,E2 6382.832} C_VEL
LIN {X 0,Y 232.5,Z 830.849,A -85,B 0,C 180,E1 6378.085,E2 6378.085} C_VEL
LIN {X 0,Y 233.336,Z 826.136,A -85,B 0,C 180,E1 6372.8,E2 6372.8} C_VEL
LIN {X 0,Y 235.238,Z 820,A -85,B 0,C 180,E1 6367.77,E2 6367.77} C_VEL
LIN {X 0,Y 238.645,Z 811.735,A -85,B 0,C 180,E1 6362.554,E2 6362.554} C_VEL
LIN {X 0,Y 243.638,Z 801.554,A -85,B 0,C 180,E1 6357.477,E2 6357.477} C_VEL
LIN {X 0,Y 249.552,Z 790.525,A -85,B 0,C 180,E1 6353.057,E2 6353.057} C_VEL
LIN {X 0,Y 256.783,Z 777.379,A -85,B 0,C 180,E1 6348.846,E2 6348.846} C_VEL
LIN {X 0,Y 264.797,Z 762.775,A -85,B 0,C 180,E1 6345.079,E2 6345.079} C_VEL
LIN {X 0,Y 273.422,Z 746.612,A -85,B 0,C 180,E1 6341.726,E2 6341.726} C_VEL
LIN {X 0,Y 281.68,Z 730.241,A -85,B 0,C 180,E1 6338.977,E2 6338.977} C_VEL
LIN {X 0,Y 290.034,Z 712.236,A -85,B 0,C 180,E1 6336.557,E2 6336.557} C_VEL
LIN {X 0,Y 297.731,Z 693.876,A -85,B 0,C 180,E1 6334.581,E2 6334.581} C_VEL
LIN {X 0,Y 305.171,Z 673.985,A -85,B 0,C 180,E1 6332.871,E2 6332.871} C_VEL
LIN {X 0,Y 311.476,Z 654.469,A -85,B 0,C 180,E1 6331.551,E2 6331.551} C_VEL
LIN {X 0,Y 316.845,Z 634.296,A -85,B 0,C 180,E1 6330.512,E2 6330.512} C_VEL
LIN {X 0,Y 321.547,Z 612.146,A -85,B 0,C 180,E1 6329.664,E2 6329.664} C_VEL
LIN {X 0,Y 324.786,Z 590.051,A -85,B 0,C 180,E1 6329.03,E2 6329.03} C_VEL
LIN {X 0,Y 340.382,Z 412.906,A -85,B 0,C 180,E1 6325.209,E2 6325.209} C_VEL
LIN {X 0,Y 336.761,Z 405.079,A -85,B 0,C 180,E1 6322.936,E2 6322.936} C_VEL
LIN {X 0,Y 333.509,Z 398.435,A -85,B 0,C 180,E1 6320.444,E2 6320.444} C_VEL
LIN {X 0,Y 331.343,Z 394.401,A -85,B 0,C 180,E1 6318.382,E2 6318.382} C_VEL
LIN {X 0,Y 330.245,Z 392.222,A -85,B 0,C 180,E1 6317.08,E2 6317.08} C_VEL
LIN {X 0,Y 328.363,Z 388.434,A -85,B 0,C 180,E1 6313.741,E2 6313.741} C_VEL
LIN {X 0,Y 327.657,Z 387.739,A -85,B 0,C 180,E1 6310.018,E2 6310.018} C_VEL
LIN {X 0,Y 328.3,Z 388.713,A -85,B 0,C 180,E1 6306.999,E2 6306.999} C_VEL
LIN {X 0,Y 330.377,Z 393.08,A -85,B 0,C 180,E1 6303.385,E2 6303.385} C_VEL
LIN {X 0,Y 332.907,Z 398.152,A -85,B 0,C 180,E1 6300.69,E2 6300.69} C_VEL
LIN {X 0,Y 336.032,Z 404.723,A -85,B 0,C 180,E1 6298.168,E2 6298.168} C_VEL
LIN {X 0,Y 339.39,Z 412.162,A -85,B 0,C 180,E1 6295.942,E2 6295.942} C_VEL
LIN {X 0,Y 323.094,Z 579.588,A -85,B 0,C 180,E1 6292.249,E2 6292.249} C_VEL
LIN {X 0,Y 319.793,Z 600.384,A -85,B 0,C 180,E1 6291.537,E2 6291.537} C_VEL
LIN {X 0,Y 315.482,Z 620.504,A -85,B 0,C 180,E1 6290.592,E2 6290.592} C_VEL
LIN {X 0,Y 310.05,Z 640.599,A -85,B 0,C 180,E1 6289.354,E2 6289.354} C_VEL
LIN {X 0,Y 304.179,Z 658.706,A -85,B 0,C 180,E1 6287.94,E2 6287.94} C_VEL
LIN {X 0,Y 297.131,Z 677.092,A -85,B 0,C 180,E1 6286.129,E2 6286.129} C_VEL
LIN {X 0,Y 289.61,Z 694.325,A -85,B 0,C 180,E1 6284.019,E2 6284.019} C_VEL
LIN {X 0,Y 281.541,Z 710.898,A -85,B 0,C 180,E1 6281.486,E2 6281.486} C_VEL
LIN {X 0,Y 273.678,Z 725.665,A -85,B 0,C 180,E1 6278.693,E2 6278.693} C_VEL
LIN {X 0,Y 265.888,Z 739.239,A -85,B 0,C 180,E1 6275.513,E2 6275.513} C_VEL
LIN {X 0,Y 257.914,Z 752.302,A -85,B 0,C 180,E1 6271.648,E2 6271.648} C_VEL
LIN {X 0,Y 251.07,Z 763.063,A -85,B 0,C 180,E1 6267.597,E2 6267.597} C_VEL
LIN {X 0,Y 245.072,Z 772.423,A -85,B 0,C 180,E1 6263.1,E2 6263.1} C_VEL
LIN {X 0,Y 240.163,Z 780.25,A -85,B 0,C 180,E1 6258.181,E2 6258.181} C_VEL
LIN {X 0,Y 236.702,Z 786.112,A -85,B 0,C 180,E1 6253.184,E2 6253.184} C_VEL
LIN {X 0,Y 234.53,Z 790.222,A -85,B 0,C 180,E1 6248.185,E2 6248.185} C_VEL
LIN {X 0,Y 233.377,Z 792.619,A -85,B 0,C 180,E1 6243.259,E2 6243.259} C_VEL
LIN {X 0,Y 232.917,Z 793.58,A -85,B 0,C 180,E1 6238.362,E2 6238.362} C_VEL
LIN {X 0,Y 232.87,Z 793.266,A -85,B 0,C 180,E1 6233.806,E2 6233.806} C_VEL
LIN {X 0,Y 233.194,Z 791.481,A -85,B 0,C 180,E1 6229.02,E2 6229.02} C_VEL
LIN {X 0,Y 234.223,Z 787.989,A -85,B 0,C 180,E1 6223.833,E2 6223.833} C_VEL
LIN {X 0,Y 236.229,Z 782.846,A -85,B 0,C 180,E1 6218.767,E2 6218.767} C_VEL
LIN {X 0,Y 239.193,Z 776.382,A -85,B 0,C 180,E1 6214.077,E2 6214.077} C_VEL
LIN {X 0,Y 243.509,Z 767.672,A -85,B 0,C 180,E1 6209.297,E2 6209.297} C_VEL
LIN {X 0,Y 248.772,Z 757.465,A -85,B 0,C 180,E1 6204.93,E2 6204.93} C_VEL
LIN {X 0,Y 254.793,Z 745.843,A -85,B 0,C 180,E1 6200.972,E2 6200.972} C_VEL
LIN {X 0,Y 261.354,Z 732.838,A -85,B 0,C 180,E1 6197.407,E2 6197.407} C_VEL
LIN {X 0,Y 268.282,Z 718.438,A -85,B 0,C 180,E1 6194.215,E2 6194.215} C_VEL
LIN {X 0,Y 275.387,Z 702.559,A -85,B 0,C 180,E1 6191.366,E2 6191.366} C_VEL
LIN {X 0,Y 282.481,Z 685.02,A -85,B 0,C 180,E1 6188.839,E2 6188.839} C_VEL
LIN {X 0,Y 288.932,Z 667.08,A -85,B 0,C 180,E1 6186.768,E2 6186.768} C_VEL
LIN {X 0,Y 294.805,Z 648.318,A -85,B 0,C 180,E1 6185.026,E2 6185.026} C_VEL
LIN {X 0,Y 300.27,Z 627.523,A -85,B 0,C 180,E1 6183.502,E2 6183.502} C_VEL
LIN {X 0,Y 304.693,Z 606.624,A -85,B 0,C 180,E1 6182.335,E2 6182.335} C_VEL
LIN {X 0,Y 308.099,Z 585.503,A -85,B 0,C 180,E1 6181.47,E2 6181.47} C_VEL
LIN {X 0,Y 310.468,Z 563.325,A -85,B 0,C 180,E1 6180.849,E2 6180.849} C_VEL
LIN {X 0,Y 322.935,Z 403.387,A -85,B 0,C 180,E1 6177.348,E2 6177.348} C_VEL
LIN {X 0,Y 314.728,Z 388.878,A -85,B 0,C 180,E1 6174.243,E2 6174.243} C_VEL
LIN {X 0,Y 306.225,Z 375.098,A -85,B 0,C 180,E1 6170.622,E2 6170.622} C_VEL
LIN {X 0,Y 298.755,Z 363.91,A -85,B 0,C 180,E1 6166.975,E2 6166.975} C_VEL
LIN {X 0,Y 292.342,Z 354.87,A -85,B 0,C 180,E1 6163.358,E2 6163.358} C_VEL
LIN {X 0,Y 289.39,Z 350.734,A -85,B 0,C 180,E1 6161.467,E2 6161.467} C_VEL
LIN {X 0,Y 287.537,Z 349.026,A -85,B 0,C 180,E1 6160.248,E2 6160.248} C_VEL
LIN {X 0,Y 284.324,Z 348.83,A -85,B 0,C 180,E1 6158.216,E2 6158.216} C_VEL
LIN {X 0,Y 281.051,Z 348.894,A -85,B 0,C 180,E1 6155.909,E2 6155.909} C_VEL
LIN {X 0,Y 279.601,Z 347.488,A -85,B 0,C 180,E1 6154.605,E2 6154.605} C_VEL
LIN {X 0,Y 275.017,Z 341.638,A -85,B 0,C 180,E1 6149.391,E2 6149.391} C_VEL
LIN {X 0,Y 271.075,Z 336.594,A -85,B 0,C 180,E1 6141.415,E2 6141.415} C_VEL
LIN {X 0,Y 270.366,Z 335.941,A -85,B 0,C 180,E1 6136.321,E2 6136.321} C_VEL
LIN {X 0,Y 271.121,Z 336.587,A -85,B 0,C 180,E1 6131.209,E2 6131.209} C_VEL
LIN {X 0,Y 274.405,Z 341.009,A -85,B 0,C 180,E1 6124.177,E2 6124.177} C_VEL
LIN {X 0,Y 275.926,Z 342.717,A -85,B 0,C 180,E1 6122.075,E2 6122.075} C_VEL
LIN {X 0,Y 280.259,Z 348.218,A -85,B 0,C 180,E1 6117.442,E2 6117.442} C_VEL
LIN {X 0,Y 284.712,Z 354.114,A -85,B 0,C 180,E1 6113.698,E2 6113.698} C_VEL
LIN {X 0,Y 289.227,Z 360.247,A -85,B 0,C 180,E1 6110.497,E2 6110.497} C_VEL
LIN {X 0,Y 294.892,Z 368.029,A -85,B 0,C 180,E1 6107.067,E2 6107.067} C_VEL
LIN {X 0,Y 301.972,Z 378.425,A -85,B 0,C 180,E1 6103.356,E2 6103.356} C_VEL
LIN {X 0,Y 309.404,Z 389.897,A -85,B 0,C 180,E1 6099.967,E2 6099.967} C_VEL
LIN {X 0,Y 317.656,Z 403.562,A -85,B 0,C 180,E1 6096.633,E2 6096.633} C_VEL
LIN {X 0,Y 322.753,Z 412.786,A -85,B 0,C 180,E1 6094.743,E2 6094.743} C_VEL
LIN {X 0,Y 308.959,Z 596.067,A -85,B 0,C 180,E1 6090.803,E2 6090.803} C_VEL
LIN {X 0,Y 305.786,Z 618.165,A -85,B 0,C 180,E1 6090.117,E2 6090.117} C_VEL
LIN {X 0,Y 301.425,Z 639.56,A -85,B 0,C 180,E1 6089.214,E2 6089.214} C_VEL
LIN {X 0,Y 296.288,Z 659.849,A -85,B 0,C 180,E1 6088.067,E2 6088.067} C_VEL
LIN {X 0,Y 290.33,Z 679.56,A -85,B 0,C 180,E1 6086.626,E2 6086.626} C_VEL
LIN {X 0,Y 283.624,Z 698.516,A -85,B 0,C 180,E1 6084.867,E2 6084.867} C_VEL
LIN {X 0,Y 276.05,Z 717.58,A -85,B 0,C 180,E1 6082.654,E2 6082.654} C_VEL
LIN {X 0,Y 268.439,Z 734.902,A -85,B 0,C 180,E1 6080.158,E2 6080.158} C_VEL
LIN {X 0,Y 260.456,Z 751.655,A -85,B 0,C 180,E1 6077.153,E2 6077.153} C_VEL
LIN {X 0,Y 252.839,Z 766.729,A -85,B 0,C 180,E1 6073.788,E2 6073.788} C_VEL
LIN {X 0,Y 245.301,Z 781.216,A -85,B 0,C 180,E1 6069.784,E2 6069.784} C_VEL
LIN {X 0,Y 238.953,Z 793.5,A -85,B 0,C 180,E1 6065.561,E2 6065.561} C_VEL
LIN {X 0,Y 233.548,Z 804.372,A -85,B 0,C 180,E1 6060.91,E2 6060.91} C_VEL
LIN {X 0,Y 229.306,Z 813.733,A -85,B 0,C 180,E1 6055.848,E2 6055.848} C_VEL
LIN {X 0,Y 226.391,Z 821.58,A -85,B 0,C 180,E1 6050.417,E2 6050.417} C_VEL
LIN {X 0,Y 224.918,Z 827.326,A -85,B 0,C 180,E1 6045.202,E2 6045.202} C_VEL
LIN {X 0,Y 224.463,Z 831.24,A -85,B 0,C 180,E1 6040.116,E2 6040.116} C_VEL
LIN {X 0,Y 224.568,Z 833.676,A -85,B 0,C 180,E1 6035.106,E2 6035.106} C_VEL
LIN {X 0,Y 224.696,Z 834.489,A -85,B 0,C 180,E1 6031.017,E2 6031.017} C_VEL
LIN {X 0,Y 224.636,Z 834.302,A -85,B 0,C 180,E1 6026.936,E2 6026.936} C_VEL
LIN {X 0,Y 224.451,Z 832.902,A -85,B 0,C 180,E1 6022.317,E2 6022.317} C_VEL
LIN {X 0,Y 224.561,Z 829.976,A -85,B 0,C 180,E1 6017.396,E2 6017.396} C_VEL
LIN {X 0,Y 225.561,Z 825.187,A -85,B 0,C 180,E1 6011.921,E2 6011.921} C_VEL
LIN {X 0,Y 227.879,Z 818.674,A -85,B 0,C 180,E1 6006.464,E2 6006.464} C_VEL
LIN {X 0,Y 231.724,Z 810.243,A -85,B 0,C 180,E1 6001.099,E2 6001.099} C_VEL
LIN {X 0,Y 237.233,Z 799.878,A -85,B 0,C 180,E1 5995.904,E2 5995.904} C_VEL
LIN {X 0,Y 244.052,Z 788.014,A -85,B 0,C 180,E1 5991.181,E2 5991.181} C_VEL
LIN {X 0,Y 252,Z 774.507,A -85,B 0,C 180,E1 5986.893,E2 5986.893} C_VEL
LIN {X 0,Y 260.004,Z 760.618,A -85,B 0,C 180,E1 5983.378,E2 5983.378} C_VEL
LIN {X 0,Y 268.782,Z 744.826,A -85,B 0,C 180,E1 5980.139,E2 5980.139} C_VEL
LIN {X 0,Y 277.602,Z 727.959,A -85,B 0,C 180,E1 5977.357,E2 5977.357} C_VEL
LIN {X 0,Y 286.603,Z 709.269,A -85,B 0,C 180,E1 5974.901,E2 5974.901} C_VEL
LIN {X 0,Y 294.465,Z 690.941,A -85,B 0,C 180,E1 5972.995,E2 5972.995} C_VEL
LIN {X 0,Y 301.694,Z 671.88,A -85,B 0,C 180,E1 5971.415,E2 5971.415} C_VEL
LIN {X 0,Y 308.119,Z 652.427,A -85,B 0,C 180,E1 5970.137,E2 5970.137} C_VEL
LIN {X 0,Y 313.632,Z 632.209,A -85,B 0,C 180,E1 5969.128,E2 5969.128} C_VEL
LIN {X 0,Y 318.218,Z 610.742,A -85,B 0,C 180,E1 5968.332,E2 5968.332} C_VEL
LIN {X 0,Y 321.6,Z 587.519,A -85,B 0,C 180,E1 5967.686,E2 5967.686} C_VEL
LIN {X 0,Y 337.19,Z 417.463,A -85,B 0,C 180,E1 5964.021,E2 5964.021} C_VEL
LIN {X 0,Y 333.569,Z 409.412,A -85,B 0,C 180,E1 5961.451,E2 5961.451} C_VEL
LIN {X 0,Y 330.778,Z 403.608,A -85,B 0,C 180,E1 5958.963,E2 5958.963} C_VEL
LIN {X 0,Y 328.885,Z 399.88,A -85,B 0,C 180,E1 5956.731,E2 5956.731} C_VEL
LIN {X 0,Y 327.162,Z 396.253,A -85,B 0,C 180,E1 5953.432,E2 5953.432} C_VEL
LIN {X 0,Y 326.604,Z 395.696,A -85,B 0,C 180,E1 5949.673,E2 5949.673} C_VEL
LIN {X 0,Y 327.147,Z 396.559,A -85,B 0,C 180,E1 5947.2,E2 5947.2} C_VEL
LIN {X 0,Y 329.043,Z 400.839,A -85,B 0,C 180,E1 5943.66,E2 5943.66} C_VEL
LIN {X 0,Y 331.36,Z 405.749,A -85,B 0,C 180,E1 5941.039,E2 5941.039} C_VEL
LIN {X 0,Y 334.581,Z 412.858,A -85,B 0,C 180,E1 5938.332,E2 5938.332} C_VEL
LIN {X 0,Y 336.232,Z 417.035,A -85,B 0,C 180,E1 5937.122,E2 5937.122} C_VEL
LIN {X 0,Y 319.758,Z 580.346,A -85,B 0,C 180,E1 5933.538,E2 5933.538} C_VEL
LIN {X 0,Y 316.357,Z 601.108,A -85,B 0,C 180,E1 5932.833,E2 5932.833} C_VEL
LIN {X 0,Y 311.886,Z 621.235,A -85,B 0,C 180,E1 5931.893,E2 5931.893} C_VEL
LIN {X 0,Y 306.268,Z 641.245,A -85,B 0,C 180,E1 5930.667,E2 5930.667} C_VEL
LIN {X 0,Y 299.803,Z 660.333,A -85,B 0,C 180,E1 5929.173,E2 5929.173} C_VEL
LIN {X 0,Y 292.527,Z 678.616,A -85,B 0,C 180,E1 5927.366,E2 5927.366} C_VEL
LIN {X 0,Y 284.812,Z 695.47,A -85,B 0,C 180,E1 5925.284,E2 5925.284} C_VEL
LIN {X 0,Y 276.415,Z 711.992,A -85,B 0,C 180,E1 5922.742,E2 5922.742} C_VEL
LIN {X 0,Y 267.911,Z 727.171,A -85,B 0,C 180,E1 5919.825,E2 5919.825} C_VEL
LIN {X 0,Y 259.513,Z 741.036,A -85,B 0,C 180,E1 5916.492,E2 5916.492} C_VEL
LIN {X 0,Y 251.524,Z 753.47,A -85,B 0,C 180,E1 5912.721,E2 5912.721} C_VEL
LIN {X 0,Y 243.967,Z 764.683,A -85,B 0,C 180,E1 5908.362,E2 5908.362} C_VEL
LIN {X 0,Y 237.794,Z 773.697,A -85,B 0,C 180,E1 5903.837,E2 5903.837} C_VEL
LIN {X 0,Y 232.732,Z 781.209,A -85,B 0,C 180,E1 5898.908,E2 5898.908} C_VEL
LIN {X 0,Y 228.961,Z 787.117,A -85,B 0,C 180,E1 5893.631,E2 5893.631} C_VEL
LIN {X 0,Y 226.652,Z 791.112,A -85,B 0,C 180,E1 5888.466,E2 5888.466} C_VEL
LIN {X 0,Y 225.433,Z 793.451,A -85,B 0,C 180,E1 5883.368,E2 5883.368} C_VEL
LIN {X 0,Y 224.949,Z 794.317,A -85,B 0,C 180,E1 5878.355,E2 5878.355} C_VEL
LIN {X 0,Y 224.906,Z 793.925,A -85,B 0,C 180,E1 5873.588,E2 5873.588} C_VEL
LIN {X 0,Y 225.275,Z 792.088,A -85,B 0,C 180,E1 5868.639,E2 5868.639} C_VEL
LIN {X 0,Y 226.332,Z 788.734,A -85,B 0,C 180,E1 5863.543,E2 5863.543} C_VEL
LIN {X 0,Y 228.462,Z 783.603,A -85,B 0,C 180,E1 5858.306,E2 5858.306} C_VEL
LIN {X 0,Y 231.598,Z 777.148,A -85,B 0,C 180,E1 5853.468,E2 5853.468} C_VEL
LIN {X 0,Y 236.151,Z 768.448,A -85,B 0,C 180,E1 5848.547,E2 5848.547} C_VEL
LIN {X 0,Y 241.68,Z 758.259,A -85,B 0,C 180,E1 5844.066,E2 5844.066} C_VEL
LIN {X 0,Y 247.984,Z 746.658,A -85,B 0,C 180,E1 5840.019,E2 5840.019} C_VEL
LIN {X 0,Y 255.258,Z 732.84,A -85,B 0,C 180,E1 5836.179,E2 5836.179} C_VEL
LIN {X 0,Y 262.507,Z 718.297,A -85,B 0,C 180,E1 5832.948,E2 5832.948} C_VEL
LIN {X 0,Y 269.649,Z 702.872,A -85,B 0,C 180,E1 5830.169,E2 5830.169} C_VEL
LIN {X 0,Y 277.022,Z 685.248,A -85,B 0,C 180,E1 5827.62,E2 5827.62} C_VEL
LIN {X 0,Y 283.697,Z 667.22,A -85,B 0,C 180,E1 5825.539,E2 5825.539} C_VEL
LIN {X 0,Y 289.766,Z 648.364,A -85,B 0,C 180,E1 5823.792,E2 5823.792} C_VEL
LIN {X 0,Y 295.277,Z 627.969,A -85,B 0,C 180,E1 5822.3,E2 5822.3} C_VEL
LIN {X 0,Y 299.854,Z 606.966,A -85,B 0,C 180,E1 5821.128,E2 5821.128} C_VEL
LIN {X 0,Y 303.355,Z 585.838,A -85,B 0,C 180,E1 5820.264,E2 5820.264} C_VEL
LIN {X 0,Y 305.794,Z 563.652,A -85,B 0,C 180,E1 5819.643,E2 5819.643} C_VEL
LIN {X 0,Y 318.3,Z 407.133,A -85,B 0,C 180,E1 5816.183,E2 5816.183} C_VEL
LIN {X 0,Y 310.711,Z 393.715,A -85,B 0,C 180,E1 5813.171,E2 5813.171} C_VEL
LIN {X 0,Y 302.89,Z 380.825,A -85,B 0,C 180,E1 5809.685,E2 5809.685} C_VEL
LIN {X 0,Y 295.869,Z 370.258,A -85,B 0,C 180,E1 5806.115,E2 5806.115} C_VEL
LIN {X 0,Y 290.408,Z 362.284,A -85,B 0,C 180,E1 5802.906,E2 5802.906} C_VEL
LIN {X 0,Y 286.552,Z 357.021,A -85,B 0,C 180,E1 5800.332,E2 5800.332} C_VEL
LIN {X 0,Y 282.906,Z 352.052,A -85,B 0,C 180,E1 5797.562,E2 5797.562} C_VEL
LIN {X 0,Y 279.601,Z 347.488,A -85,B 0,C 180,E1 5794.605,E2 5794.605} C_VEL
LIN {X 0,Y 278.641,Z 346.922,A -85,B 0,C 180,E1 5793.721,E2 5793.721} C_VEL
LIN {X 0,Y 276.781,Z 348.549,A -85,B 0,C 180,E1 5792.233,E2 5792.233} C_VEL
LIN {X 0,Y 275.023,Z 350.36,A -85,B 0,C 180,E1 5790.719,E2 5790.719} C_VEL
LIN {X 0,Y 274.219,Z 350.044,A -85,B 0,C 180,E1 5789.793,E2 5789.793} C_VEL
LIN {X 0,Y 270.094,Z 344.683,A -85,B 0,C 180,E1 5781.701,E2 5781.701} C_VEL
LIN {X 0,Y 269.351,Z 343.891,A -85,B 0,C 180,E1 5777.453,E2 5777.453} C_VEL
LIN {X 0,Y 269.847,Z 344.308,A -85,B 0,C 180,E1 5771.974,E2 5771.974} C_VEL
LIN {X 0,Y 270.856,Z 345.951,A -85,B 0,C 180,E1 5768.703,E2 5768.703} C_VEL
LIN {X 0,Y 274.518,Z 350.319,A -85,B 0,C 180,E1 5762.503,E2 5762.503} C_VEL
LIN {X 0,Y 278.828,Z 356.014,A -85,B 0,C 180,E1 5757.738,E2 5757.738} C_VEL
LIN {X 0,Y 283.012,Z 361.666,A -85,B 0,C 180,E1 5754.118,E2 5754.118} C_VEL
LIN {X 0,Y 287.455,Z 367.821,A -85,B 0,C 180,E1 5750.892,E2 5750.892} C_VEL
LIN {X 0,Y 292.786,Z 375.319,A -85,B 0,C 180,E1 5747.575,E2 5747.575} C_VEL
LIN {X 0,Y 299.763,Z 385.761,A -85,B 0,C 180,E1 5743.827,E2 5743.827} C_VEL
LIN {X 0,Y 306.786,Z 396.849,A -85,B 0,C 180,E1 5740.533,E2 5740.533} C_VEL
LIN {X 0,Y 314.796,Z 410.374,A -85,B 0,C 180,E1 5737.2,E2 5737.2} C_VEL
LIN {X 0,Y 318.199,Z 416.827,A -85,B 0,C 180,E1 5735.874,E2 5735.874} C_VEL
LIN {X 0,Y 304.329,Z 595.596,A -85,B 0,C 180,E1 5732.031,E2 5732.031} C_VEL
LIN {X 0,Y 301.101,Z 617.588,A -85,B 0,C 180,E1 5731.348,E2 5731.348} C_VEL
LIN {X 0,Y 296.735,Z 638.561,A -85,B 0,C 180,E1 5730.475,E2 5730.475} C_VEL
LIN {X 0,Y 291.285,Z 659.548,A -85,B 0,C 180,E1 5729.296,E2 5729.296} C_VEL
LIN {X 0,Y 285.16,Z 679.227,A -85,B 0,C 180,E1 5727.857,E2 5727.857} C_VEL
LIN {X 0,Y 278.257,Z 698.145,A -85,B 0,C 180,E1 5726.099,E2 5726.099} C_VEL
LIN {X 0,Y 270.445,Z 717.191,A -85,B 0,C 180,E1 5723.878,E2 5723.878} C_VEL
LIN {X 0,Y 262.771,Z 734.114,A -85,B 0,C 180,E1 5721.434,E2 5721.434} C_VEL
LIN {X 0,Y 254.823,Z 750.224,A -85,B 0,C 180,E1 5718.537,E2 5718.537} C_VEL
LIN {X 0,Y 246.832,Z 765.43,A -85,B 0,C 180,E1 5715.14,E2 5715.14} C_VEL
LIN {X 0,Y 238.907,Z 780.03,A -85,B 0,C 180,E1 5711.073,E2 5711.073} C_VEL
LIN {X 0,Y 232.176,Z 792.421,A -85,B 0,C 180,E1 5706.766,E2 5706.766} C_VEL
LIN {X 0,Y 226.403,Z 803.355,A -85,B 0,C 180,E1 5701.999,E2 5701.999} C_VEL
LIN {X 0,Y 221.874,Z 812.707,A -85,B 0,C 180,E1 5696.837,E2 5696.837} C_VEL
LIN {X 0,Y 218.629,Z 820.794,A -85,B 0,C 180,E1 5691.096,E2 5691.096} C_VEL
LIN {X 0,Y 216.994,Z 826.624,A -85,B 0,C 180,E1 5685.624,E2 5685.624} C_VEL
LIN {X 0,Y 216.488,Z 830.526,A -85,B 0,C 180,E1 5680.374,E2 5680.374} C_VEL
LIN {X 0,Y 216.586,Z 832.931,A -85,B 0,C 180,E1 5675.295,E2 5675.295} C_VEL
LIN {X 0,Y 216.728,Z 833.762,A -85,B 0,C 180,E1 5671.055,E2 5671.055} C_VEL
LIN {X 0,Y 216.671,Z 833.625,A -85,B 0,C 180,E1 5667.088,E2 5667.088} C_VEL
LIN {X 0,Y 216.469,Z 832.333,A -85,B 0,C 180,E1 5662.299,E2 5662.299} C_VEL
LIN {X 0,Y 216.585,Z 829.473,A -85,B 0,C 180,E1 5657.195,E2 5657.195} C_VEL
LIN {X 0,Y 217.659,Z 824.806,A -85,B 0,C 180,E1 5651.518,E2 5651.518} C_VEL
LIN {X 0,Y 220.136,Z 818.361,A -85,B 0,C 180,E1 5645.869,E2 5645.869} C_VEL
LIN {X 0,Y 224.22,Z 810.068,A -85,B 0,C 180,E1 5640.329,E2 5640.329} C_VEL
LIN {X 0,Y 230.042,Z 799.864,A -85,B 0,C 180,E1 5634.987,E2 5634.987} C_VEL
LIN {X 0,Y 237.213,Z 788.177,A -85,B 0,C 180,E1 5630.154,E2 5630.154} C_VEL
LIN {X 0,Y 245.419,Z 774.969,A -85,B 0,C 180,E1 5625.837,E2 5625.837} C_VEL
LIN {X 0,Y 253.859,Z 761.122,A -85,B 0,C 180,E1 5622.226,E2 5622.226} C_VEL
LIN {X 0,Y 263.257,Z 745.061,A -85,B 0,C 180,E1 5618.865,E2 5618.865} C_VEL
LIN {X 0,Y 272.293,Z 728.658,A -85,B 0,C 180,E1 5616.112,E2 5616.112} C_VEL
LIN {X 0,Y 281.309,Z 710.699,A -85,B 0,C 180,E1 5613.723,E2 5613.723} C_VEL
LIN {X 0,Y 289.448,Z 692.689,A -85,B 0,C 180,E1 5611.81,E2 5611.81} C_VEL
LIN {X 0,Y 297.233,Z 673.273,A -85,B 0,C 180,E1 5610.169,E2 5610.169} C_VEL
LIN {X 0,Y 303.816,Z 654.192,A -85,B 0,C 180,E1 5608.904,E2 5608.904} C_VEL
LIN {X 0,Y 309.456,Z 634.598,A -85,B 0,C 180,E1 5607.907,E2 5607.907} C_VEL
LIN {X 0,Y 314.537,Z 612.476,A -85,B 0,C 180,E1 5607.068,E2 5607.068} C_VEL
LIN {X 0,Y 318.055,Z 590.716,A -85,B 0,C 180,E1 5606.443,E2 5606.443} C_VEL
LIN {X 0,Y 334.179,Z 422.271,A -85,B 0,C 180,E1 5602.824,E2 5602.824} C_VEL
LIN {X 0,Y 330.92,Z 414.752,A -85,B 0,C 180,E1 5600.195,E2 5600.195} C_VEL
LIN {X 0,Y 328.909,Z 410.448,A -85,B 0,C 180,E1 5598.156,E2 5598.156} C_VEL
LIN {X 0,Y 327.499,Z 407.466,A -85,B 0,C 180,E1 5596.314,E2 5596.314} C_VEL
LIN {X 0,Y 326.037,Z 404.144,A -85,B 0,C 180,E1 5593.298,E2 5593.298} C_VEL
LIN {X 0,Y 325.541,Z 403.639,A -85,B 0,C 180,E1 5589.548,E2 5589.548} C_VEL
LIN {X 0,Y 326.02,Z 404.51,A -85,B 0,C 180,E1 5587.313,E2 5587.313} C_VEL
LIN {X 0,Y 327.659,Z 408.435,A -85,B 0,C 180,E1 5584.026,E2 5584.026} C_VEL
LIN {X 0,Y 329.932,Z 413.534,A -85,B 0,C 180,E1 5581.304,E2 5581.304} C_VEL
LIN {X 0,Y 333.006,Z 420.902,A -85,B 0,C 180,E1 5578.576,E2 5578.576} C_VEL
LIN {X 0,Y 333.301,Z 421.877,A -85,B 0,C 180,E1 5578.33,E2 5578.33} C_VEL
LIN {X 0,Y 316.716,Z 580.777,A -85,B 0,C 180,E1 5574.869,E2 5574.869} C_VEL
LIN {X 0,Y 313.183,Z 601.613,A -85,B 0,C 180,E1 5574.169,E2 5574.169} C_VEL
LIN {X 0,Y 308.648,Z 621.383,A -85,B 0,C 180,E1 5573.258,E2 5573.258} C_VEL
LIN {X 0,Y 302.763,Z 641.733,A -85,B 0,C 180,E1 5572.029,E2 5572.029} C_VEL
LIN {X 0,Y 296.425,Z 659.991,A -85,B 0,C 180,E1 5570.625,E2 5570.625} C_VEL
LIN {X 0,Y 288.796,Z 678.486,A -85,B 0,C 180,E1 5568.823,E2 5568.823} C_VEL
LIN {X 0,Y 280.512,Z 696.016,A -85,B 0,C 180,E1 5566.682,E2 5566.682} C_VEL
LIN {X 0,Y 271.797,Z 712.482,A -85,B 0,C 180,E1 5564.156,E2 5564.156} C_VEL
LIN {X 0,Y 262.938,Z 727.638,A -85,B 0,C 180,E1 5561.242,E2 5561.242} C_VEL
LIN {X 0,Y 254.459,Z 741.053,A -85,B 0,C 180,E1 5558.027,E2 5558.027} C_VEL
LIN {X 0,Y 245.692,Z 753.976,A -85,B 0,C 180,E1 5554.08,E2 5554.08} C_VEL
LIN {X 0,Y 238.072,Z 764.643,A -85,B 0,C 180,E1 5549.905,E2 5549.905} C_VEL
LIN {X 0,Y 231.285,Z 773.956,A -85,B 0,C 180,E1 5545.208,E2 5545.208} C_VEL
LIN {X 0,Y 225.654,Z 781.75,A -85,B 0,C 180,E1 5540.026,E2 5540.026} C_VEL
LIN {X 0,Y 221.619,Z 787.573,A -85,B 0,C 180,E1 5534.737,E2 5534.737} C_VEL
LIN {X 0,Y 219.008,Z 791.678,A -85,B 0,C 180,E1 5529.393,E2 5529.393} C_VEL
LIN {X 0,Y 217.591,Z 794.069,A -85,B 0,C 180,E1 5524.101,E2 5524.101} C_VEL
LIN {X 0,Y 217.017,Z 795.032,A -85,B 0,C 180,E1 5518.916,E2 5518.916} C_VEL
LIN {X 0,Y 216.929,Z 794.717,A -85,B 0,C 180,E1 5513.932,E2 5513.932} C_VEL
LIN {X 0,Y 217.285,Z 792.945,A -85,B 0,C 180,E1 5508.793,E2 5508.793} C_VEL
LIN {X 0,Y 218.447,Z 789.475,A -85,B 0,C 180,E1 5503.232,E2 5503.232} C_VEL
LIN {X 0,Y 220.57,Z 784.671,A -85,B 0,C 180,E1 5498.081,E2 5498.081} C_VEL
LIN {X 0,Y 224.032,Z 777.913,A -85,B 0,C 180,E1 5492.817,E2 5492.817} C_VEL
LIN {X 0,Y 228.56,Z 769.683,A -85,B 0,C 180,E1 5487.997,E2 5487.997} C_VEL
LIN {X 0,Y 234.307,Z 759.616,A -85,B 0,C 180,E1 5483.387,E2 5483.387} C_VEL
LIN {X 0,Y 240.85,Z 748.149,A -85,B 0,C 180,E1 5479.236,E2 5479.236} C_VEL
LIN {X 0,Y 247.944,Z 735.323,A -85,B 0,C 180,E1 5475.524,E2 5475.524} C_VEL
LIN {X 0,Y 255.398,Z 721.128,A -85,B 0,C 180,E1 5472.223,E2 5472.223} C_VEL
LIN {X 0,Y 263.25,Z 704.856,A -85,B 0,C 180,E1 5469.202,E2 5469.202} C_VEL
LIN {X 0,Y 270.556,Z 688.11,A -85,B 0,C 180,E1 5466.71,E2 5466.71} C_VEL
LIN {X 0,Y 277.419,Z 670.552,A -85,B 0,C 180,E1 5464.605,E2 5464.605} C_VEL
LIN {X 0,Y 283.957,Z 651.346,A -85,B 0,C 180,E1 5462.761,E2 5462.761} C_VEL
LIN {X 0,Y 289.611,Z 631.652,A -85,B 0,C 180,E1 5461.267,E2 5461.267} C_VEL
LIN {X 0,Y 294.5,Z 610.666,A -85,B 0,C 180,E1 5460.042,E2 5460.042} C_VEL
LIN {X 0,Y 298.429,Z 588.358,A -85,B 0,C 180,E1 5459.095,E2 5459.095} C_VEL
LIN {X 0,Y 301.018,Z 566.266,A -85,B 0,C 180,E1 5458.459,E2 5458.459} C_VEL
LIN {X 0,Y 313.835,Z 411.147,A -85,B 0,C 180,E1 5455.031,E2 5455.031} C_VEL
LIN {X 0,Y 306.637,Z 398.249,A -85,B 0,C 180,E1 5452.021,E2 5452.021} C_VEL
LIN {X 0,Y 299.419,Z 386.348,A -85,B 0,C 180,E1 5448.639,E2 5448.639} C_VEL
LIN {X 0,Y 292.922,Z 376.365,A -85,B 0,C 180,E1 5445.161,E2 5445.161} C_VEL
LIN {X 0,Y 288.08,Z 369.185,A -85,B 0,C 180,E1 5442.187,E2 5442.187} C_VEL
LIN {X 0,Y 284.561,Z 364.269,A -85,B 0,C 180,E1 5439.751,E2 5439.751} C_VEL
LIN {X 0,Y 281.165,Z 359.513,A -85,B 0,C 180,E1 5437.065,E2 5437.065} C_VEL
LIN {X 0,Y 277.529,Z 354.474,A -85,B 0,C 180,E1 5433.677,E2 5433.677} C_VEL
LIN {X 0,Y 274.219,Z 350.044,A -85,B 0,C 180,E1 5429.793,E2 5429.793} C_VEL
LIN {X 0,Y 273.217,Z 349.275,A -85,B 0,C 180,E1 5428.437,E2 5428.437} C_VEL
LIN {X 0,Y 271.638,Z 350.522,A -85,B 0,C 180,E1 5426.49,E2 5426.49} C_VEL
LIN {X 0,Y 269.773,Z 353.06,A -85,B 0,C 180,E1 5423.695,E2 5423.695} C_VEL
LIN {X 0,Y 269.215,Z 353.005,A -85,B 0,C 180,E1 5422.388,E2 5422.388} C_VEL
LIN {X 0,Y 268.453,Z 351.934,A -85,B 0,C 180,E1 5419.131,E2 5419.131} C_VEL
LIN {X 0,Y 268.588,Z 352.038,A -85,B 0,C 180,E1 5412.904,E2 5412.904} C_VEL
LIN {X 0,Y 269.464,Z 353.337,A -85,B 0,C 180,E1 5409.61,E2 5409.61} C_VEL
LIN {X 0,Y 273.202,Z 358.08,A -85,B 0,C 180,E1 5402.82,E2 5402.82} C_VEL
LIN {X 0,Y 277.292,Z 363.63,A -85,B 0,C 180,E1 5398.139,E2 5398.139} C_VEL
LIN {X 0,Y 281.389,Z 369.315,A -85,B 0,C 180,E1 5394.493,E2 5394.493} C_VEL
LIN {X 0,Y 285.689,Z 375.39,A -85,B 0,C 180,E1 5391.292,E2 5391.292} C_VEL
LIN {X 0,Y 290.773,Z 382.734,A -85,B 0,C 180,E1 5388.042,E2 5388.042} C_VEL
LIN {X 0,Y 297.369,Z 392.805,A -85,B 0,C 180,E1 5384.395,E2 5384.395} C_VEL
LIN {X 0,Y 304.08,Z 403.627,A -85,B 0,C 180,E1 5381.151,E2 5381.151} C_VEL
LIN {X 0,Y 311.747,Z 416.84,A -85,B 0,C 180,E1 5377.86,E2 5377.86} C_VEL
LIN {X 0,Y 313.765,Z 420.742,A -85,B 0,C 180,E1 5377.038,E2 5377.038} C_VEL
LIN {X 0,Y 299.75,Z 595.389,A -85,B 0,C 180,E1 5373.28,E2 5373.28} C_VEL
LIN {X 0,Y 296.407,Z 617.569,A -85,B 0,C 180,E1 5372.592,E2 5372.592} C_VEL
LIN {X 0,Y 291.824,Z 638.91,A -85,B 0,C 180,E1 5371.702,E2 5371.702} C_VEL
LIN {X 0,Y 286.062,Z 660.316,A -85,B 0,C 180,E1 5370.49,E2 5370.49} C_VEL
LIN {X 0,Y 279.566,Z 680.459,A -85,B 0,C 180,E1 5369,E2 5369} C_VEL
LIN {X 0,Y 272.367,Z 699.455,A -85,B 0,C 180,E1 5367.205,E2 5367.205} C_VEL
LIN {X 0,Y 264.654,Z 717.479,A -85,B 0,C 180,E1 5365.062,E2 5365.062} C_VEL
LIN {X 0,Y 256.654,Z 734.423,A -85,B 0,C 180,E1 5362.572,E2 5362.572} C_VEL
LIN {X 0,Y 248.251,Z 750.831,A -85,B 0,C 180,E1 5359.567,E2 5359.567} C_VEL
LIN {X 0,Y 239.993,Z 765.867,A -85,B 0,C 180,E1 5356.112,E2 5356.112} C_VEL
LIN {X 0,Y 232.212,Z 779.578,A -85,B 0,C 180,E1 5352.195,E2 5352.195} C_VEL
LIN {X 0,Y 225.075,Z 792.051,A -85,B 0,C 180,E1 5347.743,E2 5347.743} C_VEL
LIN {X 0,Y 219.023,Z 802.92,A -85,B 0,C 180,E1 5342.86,E2 5342.86} C_VEL
LIN {X 0,Y 214.223,Z 812.259,A -85,B 0,C 180,E1 5337.517,E2 5337.517} C_VEL
LIN {X 0,Y 210.8,Z 820.247,A -85,B 0,C 180,E1 5331.615,E2 5331.615} C_VEL
LIN {X 0,Y 209.062,Z 825.993,A -85,B 0,C 180,E1 5325.987,E2 5325.987} C_VEL
LIN {X 0,Y 208.51,Z 829.899,A -85,B 0,C 180,E1 5320.496,E2 5320.496} C_VEL
LIN {X 0,Y 208.618,Z 832.255,A -85,B 0,C 180,E1 5315.222,E2 5315.222} C_VEL
LIN {X 0,Y 208.763,Z 833.052,A -85,B 0,C 180,E1 5310.82,E2 5310.82} C_VEL
LIN {X 0,Y 208.684,Z 832.874,A -85,B 0,C 180,E1 5306.701,E2 5306.701} C_VEL
LIN {X 0,Y 208.471,Z 831.521,A -85,B 0,C 180,E1 5301.725,E2 5301.725} C_VEL
LIN {X 0,Y 208.665,Z 828.608,A -85,B 0,C 180,E1 5296.418,E2 5296.418} C_VEL
LIN {X 0,Y 209.958,Z 823.874,A -85,B 0,C 180,E1 5290.525,E2 5290.525} C_VEL
LIN {X 0,Y 212.751,Z 817.389,A -85,B 0,C 180,E1 5284.677,E2 5284.677} C_VEL
LIN {X 0,Y 217.269,Z 809.04,A -85,B 0,C 180,E1 5278.972,E2 5278.972} C_VEL
LIN {X 0,Y 223.596,Z 798.782,A -85,B 0,C 180,E1 5273.503,E2 5273.503} C_VEL
LIN {X 0,Y 230.866,Z 787.701,A -85,B 0,C 180,E1 5268.827,E2 5268.827} C_VEL
LIN {X 0,Y 239.529,Z 774.555,A -85,B 0,C 180,E1 5264.452,E2 5264.452} C_VEL
LIN {X 0,Y 248.37,Z 760.777,A -85,B 0,C 180,E1 5260.812,E2 5260.812} C_VEL
LIN {X 0,Y 258.175,Z 744.858,A -85,B 0,C 180,E1 5257.443,E2 5257.443} C_VEL
LIN {X 0,Y 267.559,Z 728.552,A -85,B 0,C 180,E1 5254.698,E2 5254.698} C_VEL
LIN {X 0,Y 276.885,Z 710.737,A -85,B 0,C 180,E1 5252.326,E2 5252.326} C_VEL
LIN {X 0,Y 285.639,Z 692.088,A -85,B 0,C 180,E1 5250.358,E2 5250.358} C_VEL
LIN {X 0,Y 293.658,Z 672.755,A -85,B 0,C 180,E1 5248.745,E2 5248.745} C_VEL
LIN {X 0,Y 300.429,Z 653.787,A -85,B 0,C 180,E1 5247.506,E2 5247.506} C_VEL
LIN {X 0,Y 306.217,Z 634.272,A -85,B 0,C 180,E1 5246.532,E2 5246.532} C_VEL
LIN {X 0,Y 311.448,Z 612.153,A -85,B 0,C 180,E1 5245.706,E2 5245.706} C_VEL
LIN {X 0,Y 315.1,Z 590.407,A -85,B 0,C 180,E1 5245.088,E2 5245.088} C_VEL
LIN {X 0,Y 331.37,Z 427.197,A -85,B 0,C 180,E1 5241.601,E2 5241.601} C_VEL
LIN {X 0,Y 328.626,Z 420.6,A -85,B 0,C 180,E1 5239.092,E2 5239.092} C_VEL
LIN {X 0,Y 326.449,Z 415.566,A -85,B 0,C 180,E1 5236.368,E2 5236.368} C_VEL
LIN {X 0,Y 324.915,Z 412.035,A -85,B 0,C 180,E1 5233.164,E2 5233.164} C_VEL
LIN {X 0,Y 324.467,Z 411.567,A -85,B 0,C 180,E1 5229.559,E2 5229.559} C_VEL
LIN {X 0,Y 324.873,Z 412.354,A -85,B 0,C 180,E1 5227.517,E2 5227.517} C_VEL
LIN {X 0,Y 326.344,Z 416.192,A -85,B 0,C 180,E1 5224.306,E2 5224.306} C_VEL
LIN {X 0,Y 328.345,Z 420.964,A -85,B 0,C 180,E1 5221.746,E2 5221.746} C_VEL
LIN {X 0,Y 330.57,Z 426.785,A -85,B 0,C 180,E1 5219.56,E2 5219.56} C_VEL
LIN {X 0,Y 313.893,Z 581.237,A -85,B 0,C 180,E1 5216.228,E2 5216.228} C_VEL
LIN {X 0,Y 310.245,Z 602.045,A -85,B 0,C 180,E1 5215.539,E2 5215.539} C_VEL
LIN {X 0,Y 305.574,Z 621.861,A -85,B 0,C 180,E1 5214.641,E2 5214.641} C_VEL
LIN {X 0,Y 299.819,Z 641.317,A -85,B 0,C 180,E1 5213.491,E2 5213.491} C_VEL
LIN {X 0,Y 293.244,Z 659.679,A -85,B 0,C 180,E1 5212.108,E2 5212.108} C_VEL
LIN {X 0,Y 285.298,Z 678.418,A -85,B 0,C 180,E1 5210.317,E2 5210.317} C_VEL
LIN {X 0,Y 276.796,Z 695.87,A -85,B 0,C 180,E1 5208.222,E2 5208.222} C_VEL
LIN {X 0,Y 267.355,Z 713.035,A -85,B 0,C 180,E1 5205.613,E2 5205.613} C_VEL
LIN {X 0,Y 258.495,Z 727.635,A -85,B 0,C 180,E1 5202.829,E2 5202.829} C_VEL
LIN {X 0,Y 249.286,Z 741.532,A -85,B 0,C 180,E1 5199.495,E2 5199.495} C_VEL
LIN {X 0,Y 240.339,Z 754.061,A -85,B 0,C 180,E1 5195.66,E2 5195.66} C_VEL
LIN {X 0,Y 232.231,Z 764.803,A -85,B 0,C 180,E1 5191.443,E2 5191.443} C_VEL
LIN {X 0,Y 224.959,Z 774.207,A -85,B 0,C 180,E1 5186.681,E2 5186.681} C_VEL
LIN {X 0,Y 219.089,Z 781.771,A -85,B 0,C 180,E1 5181.639,E2 5181.639} C_VEL
LIN {X 0,Y 214.583,Z 787.777,A -85,B 0,C 180,E1 5176.242,E2 5176.242} C_VEL
LIN {X 0,Y 211.411,Z 792.204,A -85,B 0,C 180,E1 5170.389,E2 5170.389} C_VEL
LIN {X 0,Y 209.771,Z 794.691,A -85,B 0,C 180,E1 5164.891,E2 5164.891} C_VEL
LIN {X 0,Y 209.065,Z 795.763,A -85,B 0,C 180,E1 5159.2,E2 5159.2} C_VEL
LIN {X 0,Y 208.961,Z 795.435,A -85,B 0,C 180,E1 5153.955,E2 5153.955} C_VEL
LIN {X 0,Y 209.331,Z 793.673,A -85,B 0,C 180,E1 5148.667,E2 5148.667} C_VEL
LIN {X 0,Y 210.567,Z 790.208,A -85,B 0,C 180,E1 5142.898,E2 5142.898} C_VEL
LIN {X 0,Y 212.824,Z 785.412,A -85,B 0,C 180,E1 5137.562,E2 5137.562} C_VEL
LIN {X 0,Y 216.492,Z 778.654,A -85,B 0,C 180,E1 5132.12,E2 5132.12} C_VEL
LIN {X 0,Y 221.273,Z 770.432,A -85,B 0,C 180,E1 5127.154,E2 5127.154} C_VEL
LIN {X 0,Y 227.317,Z 760.378,A -85,B 0,C 180,E1 5122.42,E2 5122.42} C_VEL
LIN {X 0,Y 234.169,Z 748.927,A -85,B 0,C 180,E1 5118.176,E2 5118.176} C_VEL
LIN {X 0,Y 241.574,Z 736.122,A -85,B 0,C 180,E1 5114.396,E2 5114.396} C_VEL
LIN {X 0,Y 249.326,Z 721.938,A -85,B 0,C 180,E1 5111.048,E2 5111.048} C_VEL
LIN {X 0,Y 257.193,Z 706.222,A -85,B 0,C 180,E1 5108.089,E2 5108.089} C_VEL
LIN {X 0,Y 264.738,Z 689.605,A -85,B 0,C 180,E1 5105.574,E2 5105.574} C_VEL
LIN {X 0,Y 272.112,Z 671.415,A -85,B 0,C 180,E1 5103.369,E2 5103.369} C_VEL
LIN {X 0,Y 278.852,Z 652.258,A -85,B 0,C 180,E1 5101.52,E2 5101.52} C_VEL
LIN {X 0,Y 284.518,Z 633.298,A -85,B 0,C 180,E1 5100.068,E2 5100.068} C_VEL
LIN {X 0,Y 289.641,Z 612.077,A -85,B 0,C 180,E1 5098.817,E2 5098.817} C_VEL
LIN {X 0,Y 293.61,Z 590.453,A -85,B 0,C 180,E1 5097.885,E2 5097.885} C_VEL
LIN {X 0,Y 296.312,Z 569.098,A -85,B 0,C 180,E1 5097.247,E2 5097.247} C_VEL
LIN {X 0,Y 309.52,Z 415.286,A -85,B 0,C 180,E1 5093.857,E2 5093.857} C_VEL
LIN {X 0,Y 303.107,Z 403.699,A -85,B 0,C 180,E1 5091.044,E2 5091.044} C_VEL
LIN {X 0,Y 296.79,Z 393.043,A -85,B 0,C 180,E1 5087.956,E2 5087.956} C_VEL
LIN {X 0,Y 290.499,Z 383.142,A -85,B 0,C 180,E1 5084.457,E2 5084.457} C_VEL
LIN {X 0,Y 285.805,Z 376.081,A -85,B 0,C 180,E1 5081.462,E2 5081.462} C_VEL
LIN {X 0,Y 282.703,Z 371.643,A -85,B 0,C 180,E1 5079.239,E2 5079.239} C_VEL
LIN {X 0,Y 279.428,Z 366.97,A -85,B 0,C 180,E1 5076.565,E2 5076.565} C_VEL
LIN {X 0,Y 275.917,Z 362.018,A -85,B 0,C 180,E1 5073.171,E2 5073.171} C_VEL
LIN {X 0,Y 272.373,Z 357.169,A -85,B 0,C 180,E1 5068.741,E2 5068.741} C_VEL
LIN {X 0,Y 269.215,Z 353.005,A -85,B 0,C 180,E1 5062.388,E2 5062.388} C_VEL
LIN {X 0,Y 268.698,Z 353.151,A -85,B 0,C 180,E1 5060.862,E2 5060.862} C_VEL
LIN {X 0,Y 267.835,Z 355.913,A -85,B 0,C 180,E1 5058.555,E2 5058.555} C_VEL
LIN {X 0,Y 267.256,Z 359.233,A -85,B 0,C 180,E1 5055.991,E2 5055.991} C_VEL
LIN {X 0,Y 267.247,Z 359.736,A -85,B 0,C 180,E1 5054.912,E2 5054.912} C_VEL
LIN {X 0,Y 268.061,Z 360.643,A -85,B 0,C 180,E1 5050.747,E2 5050.747} C_VEL
LIN {X 0,Y 271.95,Z 365.954,A -85,B 0,C 180,E1 5043.054,E2 5043.054} C_VEL
LIN {X 0,Y 275.77,Z 371.245,A -85,B 0,C 180,E1 5038.544,E2 5038.544} C_VEL
LIN {X 0,Y 279.778,Z 376.961,A -85,B 0,C 180,E1 5034.873,E2 5034.873} C_VEL
LIN {X 0,Y 283.906,Z 382.908,A -85,B 0,C 180,E1 5031.72,E2 5031.72} C_VEL
LIN {X 0,Y 288.933,Z 390.397,A -85,B 0,C 180,E1 5028.42,E2 5028.42} C_VEL
LIN {X 0,Y 295.174,Z 400.126,A -85,B 0,C 180,E1 5024.88,E2 5024.88} C_VEL
LIN {X 0,Y 301.584,Z 410.732,A -85,B 0,C 180,E1 5021.69,E2 5021.69} C_VEL
LIN {X 0,Y 308.813,Z 423.491,A -85,B 0,C 180,E1 5018.488,E2 5018.488} C_VEL
LIN {X 0,Y 309.4,Z 425.004,A -85,B 0,C 180,E1 5018.223,E2 5018.223} C_VEL
LIN {X 0,Y 295.35,Z 594.852,A -85,B 0,C 180,E1 5014.575,E2 5014.575} C_VEL
LIN {X 0,Y 291.962,Z 616.886,A -85,B 0,C 180,E1 5013.896,E2 5013.896} C_VEL
LIN {X 0,Y 287.237,Z 638.42,A -85,B 0,C 180,E1 5013.009,E2 5013.009} C_VEL
LIN {X 0,Y 281.328,Z 659.821,A -85,B 0,C 180,E1 5011.807,E2 5011.807} C_VEL
LIN {X 0,Y 274.88,Z 679.358,A -85,B 0,C 180,E1 5010.377,E2 5010.377} C_VEL
LIN {X 0,Y 267.25,Z 698.949,A -85,B 0,C 180,E1 5008.536,E2 5008.536} C_VEL
LIN {X 0,Y 259.299,Z 717.002,A -85,B 0,C 180,E1 5006.392,E2 5006.392} C_VEL
LIN {X 0,Y 250.936,Z 734.147,A -85,B 0,C 180,E1 5003.862,E2 5003.862} C_VEL
LIN {X 0,Y 242.266,Z 750.491,A -85,B 0,C 180,E1 5000.841,E2 5000.841} C_VEL
LIN {X 0,Y 233.729,Z 765.385,A -85,B 0,C 180,E1 4997.369,E2 4997.369} C_VEL
LIN {X 0,Y 225.585,Z 779.109,A -85,B 0,C 180,E1 4993.371,E2 4993.371} C_VEL
LIN {X 0,Y 218.188,Z 791.421,A -85,B 0,C 180,E1 4988.885,E2 4988.885} C_VEL
LIN {X 0,Y 211.67,Z 802.529,A -85,B 0,C 180,E1 4983.758,E2 4983.758} C_VEL
LIN {X 0,Y 206.617,Z 811.769,A -85,B 0,C 180,E1 4978.266,E2 4978.266} C_VEL
LIN {X 0,Y 203.035,Z 819.562,A -85,B 0,C 180,E1 4972.28,E2 4972.28} C_VEL
LIN {X 0,Y 201.137,Z 825.351,A -85,B 0,C 180,E1 4966.376,E2 4966.376} C_VEL
LIN {X 0,Y 200.538,Z 829.16,A -85,B 0,C 180,E1 4960.813,E2 4960.813} C_VEL
LIN {X 0,Y 200.635,Z 831.505,A -85,B 0,C 180,E1 4955.43,E2 4955.43} C_VEL
LIN {X 0,Y 200.796,Z 832.324,A -85,B 0,C 180,E1 4950.853,E2 4950.853} C_VEL
LIN {X 0,Y 200.708,Z 832.161,A -85,B 0,C 180,E1 4946.57,E2 4946.57} C_VEL
LIN {X 0,Y 200.482,Z 830.829,A -85,B 0,C 180,E1 4941.392,E2 4941.392} C_VEL
LIN {X 0,Y 200.731,Z 827.929,A -85,B 0,C 180,E1 4935.87,E2 4935.87} C_VEL
LIN {X 0,Y 202.187,Z 823.229,A -85,B 0,C 180,E1 4929.744,E2 4929.744} C_VEL
LIN {X 0,Y 205.275,Z 816.747,A -85,B 0,C 180,E1 4923.67,E2 4923.67} C_VEL
LIN {X 0,Y 210.167,Z 808.467,A -85,B 0,C 180,E1 4917.8,E2 4917.8} C_VEL
LIN {X 0,Y 216.946,Z 798.264,A -85,B 0,C 180,E1 4912.193,E2 4912.193} C_VEL
LIN {X 0,Y 224.656,Z 787.265,A -85,B 0,C 180,E1 4907.427,E2 4907.427} C_VEL
LIN {X 0,Y 233.788,Z 774.156,A -85,B 0,C 180,E1 4902.999,E2 4902.999} C_VEL
LIN {X 0,Y 243.179,Z 760.307,A -85,B 0,C 180,E1 4899.288,E2 4899.288} C_VEL
LIN {X 0,Y 253.263,Z 744.685,A -85,B 0,C 180,E1 4895.967,E2 4895.967} C_VEL
LIN {X 0,Y 263.002,Z 728.518,A -85,B 0,C 180,E1 4893.237,E2 4893.237} C_VEL
LIN {X 0,Y 272.636,Z 710.821,A -85,B 0,C 180,E1 4890.885,E2 4890.885} C_VEL
LIN {X 0,Y 281.658,Z 692.427,A -85,B 0,C 180,E1 4888.946,E2 4888.946} C_VEL
LIN {X 0,Y 289.897,Z 673.344,A -85,B 0,C 180,E1 4887.359,E2 4887.359} C_VEL
LIN {X 0,Y 296.837,Z 654.592,A -85,B 0,C 180,E1 4886.143,E2 4886.143} C_VEL
LIN {X 0,Y 303.166,Z 634.174,A -85,B 0,C 180,E1 4885.131,E2 4885.131} C_VEL
LIN {X 0,Y 308.394,Z 612.961,A -85,B 0,C 180,E1 4884.347,E2 4884.347} C_VEL
LIN {X 0,Y 312.289,Z 590.836,A -85,B 0,C 180,E1 4883.722,E2 4883.722} C_VEL
LIN {X 0,Y 328.761,Z 432.378,A -85,B 0,C 180,E1 4880.369,E2 4880.369} C_VEL
LIN {X 0,Y 326.483,Z 426.464,A -85,B 0,C 180,E1 4877.927,E2 4877.927} C_VEL
LIN {X 0,Y 324.929,Z 422.901,A -85,B 0,C 180,E1 4875.713,E2 4875.713} C_VEL
LIN {X 0,Y 323.793,Z 419.927,A -85,B 0,C 180,E1 4873.029,E2 4873.029} C_VEL
LIN {X 0,Y 323.406,Z 419.51,A -85,B 0,C 180,E1 4869.432,E2 4869.432} C_VEL
LIN {X 0,Y 323.751,Z 420.302,A -85,B 0,C 180,E1 4867.633,E2 4867.633} C_VEL
LIN {X 0,Y 325.037,Z 423.948,A -85,B 0,C 180,E1 4864.589,E2 4864.589} C_VEL
LIN {X 0,Y 326.777,Z 428.395,A -85,B 0,C 180,E1 4862.193,E2 4862.193} C_VEL
LIN {X 0,Y 327.993,Z 432.091,A -85,B 0,C 180,E1 4860.805,E2 4860.805} C_VEL
LIN {X 0,Y 311.282,Z 581.914,A -85,B 0,C 180,E1 4857.608,E2 4857.608} C_VEL
LIN {X 0,Y 307.526,Z 602.758,A -85,B 0,C 180,E1 4856.929,E2 4856.929} C_VEL
LIN {X 0,Y 302.579,Z 622.994,A -85,B 0,C 180,E1 4856.022,E2 4856.022} C_VEL
LIN {X 0,Y 296.182,Z 643.577,A -85,B 0,C 180,E1 4854.804,E2 4854.804} C_VEL
LIN {X 0,Y 288.919,Z 662.836,A -85,B 0,C 180,E1 4853.335,E2 4853.335} C_VEL
LIN {X 0,Y 280.978,Z 680.74,A -85,B 0,C 180,E1 4851.606,E2 4851.606} C_VEL
LIN {X 0,Y 272.453,Z 697.358,A -85,B 0,C 180,E1 4849.591,E2 4849.591} C_VEL
LIN {X 0,Y 262.814,Z 714.17,A -85,B 0,C 180,E1 4847.031,E2 4847.031} C_VEL
LIN {X 0,Y 253.148,Z 729.295,A -85,B 0,C 180,E1 4844.109,E2 4844.109} C_VEL
LIN {X 0,Y 243.584,Z 743.032,A -85,B 0,C 180,E1 4840.757,E2 4840.757} C_VEL
LIN {X 0,Y 234.246,Z 755.432,A -85,B 0,C 180,E1 4836.88,E2 4836.88} C_VEL
LIN {X 0,Y 225.706,Z 766.109,A -85,B 0,C 180,E1 4832.57,E2 4832.57} C_VEL
LIN {X 0,Y 218.337,Z 775.014,A -85,B 0,C 180,E1 4827.912,E2 4827.912} C_VEL
LIN {X 0,Y 211.789,Z 782.876,A -85,B 0,C 180,E1 4822.483,E2 4822.483} C_VEL
LIN {X 0,Y 206.953,Z 788.808,A -85,B 0,C 180,E1 4816.85,E2 4816.85} C_VEL
LIN {X 0,Y 203.59,Z 793.162,A -85,B 0,C 180,E1 4810.785,E2 4810.785} C_VEL
LIN {X 0,Y 201.843,Z 795.538,A -85,B 0,C 180,E1 4805.076,E2 4805.076} C_VEL
LIN {X 0,Y 201.117,Z 796.492,A -85,B 0,C 180,E1 4799.487,E2 4799.487} C_VEL
LIN {X 0,Y 200.988,Z 796.165,A -85,B 0,C 180,E1 4794.078,E2 4794.078} C_VEL
LIN {X 0,Y 201.381,Z 794.388,A -85,B 0,C 180,E1 4788.511,E2 4788.511} C_VEL
LIN {X 0,Y 202.694,Z 790.938,A -85,B 0,C 180,E1 4782.538,E2 4782.538} C_VEL
LIN {X 0,Y 205.096,Z 786.15,A -85,B 0,C 180,E1 4777.003,E2 4777.003} C_VEL
LIN {X 0,Y 209.016,Z 779.347,A -85,B 0,C 180,E1 4771.339,E2 4771.339} C_VEL
LIN {X 0,Y 214.037,Z 771.179,A -85,B 0,C 180,E1 4766.253,E2 4766.253} C_VEL
LIN {X 0,Y 220.393,Z 761.128,A -85,B 0,C 180,E1 4761.393,E2 4761.393} C_VEL
LIN {X 0,Y 227.998,Z 748.978,A -85,B 0,C 180,E1 4756.821,E2 4756.821} C_VEL
LIN {X 0,Y 235.774,Z 736.034,A -85,B 0,C 180,E1 4752.988,E2 4752.988} C_VEL
LIN {X 0,Y 243.88,Z 721.711,A -85,B 0,C 180,E1 4749.608,E2 4749.608} C_VEL
LIN {X 0,Y 252.367,Z 705.333,A -85,B 0,C 180,E1 4746.539,E2 4746.539} C_VEL
LIN {X 0,Y 260.277,Z 688.3,A -85,B 0,C 180,E1 4744.01,E2 4744.01} C_VEL
LIN {X 0,Y 267.559,Z 670.66,A -85,B 0,C 180,E1 4741.913,E2 4741.913} C_VEL
LIN {X 0,Y 274.521,Z 651.206,A -85,B 0,C 180,E1 4740.07,E2 4740.07} C_VEL
LIN {X 0,Y 280.355,Z 631.845,A -85,B 0,C 180,E1 4738.624,E2 4738.624} C_VEL
LIN {X 0,Y 285.458,Z 610.968,A -85,B 0,C 180,E1 4737.425,E2 4737.425} C_VEL
LIN {X 0,Y 289.569,Z 588.76,A -85,B 0,C 180,E1 4736.496,E2 4736.496} C_VEL
LIN {X 0,Y 292.325,Z 566.291,A -85,B 0,C 180,E1 4735.86,E2 4735.86} C_VEL
LIN {X 0,Y 305.257,Z 419.386,A -85,B 0,C 180,E1 4732.646,E2 4732.646} C_VEL
LIN {X 0,Y 298.202,Z 406.571,A -85,B 0,C 180,E1 4729.345,E2 4729.345} C_VEL
LIN {X 0,Y 292.161,Z 396.37,A -85,B 0,C 180,E1 4726.154,E2 4726.154} C_VEL
LIN {X 0,Y 285.948,Z 386.538,A -85,B 0,C 180,E1 4722.372,E2 4722.372} C_VEL
LIN {X 0,Y 281.067,Z 379.276,A -85,B 0,C 180,E1 4718.877,E2 4718.877} C_VEL
LIN {X 0,Y 277.833,Z 374.571,A -85,B 0,C 180,E1 4716.168,E2 4716.168} C_VEL
LIN {X 0,Y 274.518,Z 369.759,A -85,B 0,C 180,E1 4712.864,E2 4712.864} C_VEL
LIN {X 0,Y 271.064,Z 364.935,A -85,B 0,C 180,E1 4708.411,E2 4708.411} C_VEL
LIN {X 0,Y 267.791,Z 360.289,A -85,B 0,C 180,E1 4701.002,E2 4701.002} C_VEL
LIN {X 0,Y 267.209,Z 359.711,A -85,B 0,C 180,E1 4695.405,E2 4695.405} C_VEL
LIN {X 0,Y 267.247,Z 359.736,A -85,B 0,C 180,E1 4694.912,E2 4694.912} C_VEL
LIN {X 0,Y 267.323,Z 360.844,A -85,B 0,C 180,E1 4693.386,E2 4693.386} C_VEL
LIN {X 0,Y 267.352,Z 365.141,A -85,B 0,C 180,E1 4691.036,E2 4691.036} C_VEL
LIN {X 0,Y 267.743,Z 369.745,A -85,B 0,C 180,E1 4688.564,E2 4688.564} C_VEL
LIN {X 0,Y 268.111,Z 370.684,A -85,B 0,C 180,E1 4687.627,E2 4687.627} C_VEL
LIN {X 0,Y 270.638,Z 373.696,A -85,B 0,C 180,E1 4683.387,E2 4683.387} C_VEL
LIN {X 0,Y 274.358,Z 379.031,A -85,B 0,C 180,E1 4678.85,E2 4678.85} C_VEL
LIN {X 0,Y 278.064,Z 384.412,A -85,B 0,C 180,E1 4675.358,E2 4675.358} C_VEL
LIN {X 0,Y 282.134,Z 390.419,A -85,B 0,C 180,E1 4672.157,E2 4672.157} C_VEL
LIN {X 0,Y 287.031,Z 397.923,A -85,B 0,C 180,E1 4668.851,E2 4668.851} C_VEL
LIN {X 0,Y 293.513,Z 408.26,A -85,B 0,C 180,E1 4665.095,E2 4665.095} C_VEL
LIN {X 0,Y 300.699,Z 420.589,A -85,B 0,C 180,E1 4661.484,E2 4661.484} C_VEL
LIN {X 0,Y 305.156,Z 428.986,A -85,B 0,C 180,E1 4659.444,E2 4659.444} C_VEL
LIN {X 0,Y 291.019,Z 594.628,A -85,B 0,C 180,E1 4655.894,E2 4655.894} C_VEL
LIN {X 0,Y 287.546,Z 616.674,A -85,B 0,C 180,E1 4655.219,E2 4655.219} C_VEL
LIN {X 0,Y 282.804,Z 637.815,A -85,B 0,C 180,E1 4654.357,E2 4654.357} C_VEL
LIN {X 0,Y 277.122,Z 658.106,A -85,B 0,C 180,E1 4653.244,E2 4653.244} C_VEL
LIN {X 0,Y 270.493,Z 677.834,A -85,B 0,C 180,E1 4651.83,E2 4651.83} C_VEL
LIN {X 0,Y 262.981,Z 696.751,A -85,B 0,C 180,E1 4650.09,E2 4650.09} C_VEL
LIN {X 0,Y 254.402,Z 715.821,A -85,B 0,C 180,E1 4647.866,E2 4647.866} C_VEL
LIN {X 0,Y 245.639,Z 733.263,A -85,B 0,C 180,E1 4645.303,E2 4645.303} C_VEL
LIN {X 0,Y 236.529,Z 749.853,A -85,B 0,C 180,E1 4642.226,E2 4642.226} C_VEL
LIN {X 0,Y 227.586,Z 764.877,A -85,B 0,C 180,E1 4638.695,E2 4638.695} C_VEL
LIN {X 0,Y 218.969,Z 778.777,A -85,B 0,C 180,E1 4634.573,E2 4634.573} C_VEL
